KUKA KRL program: MyProgram_299().src

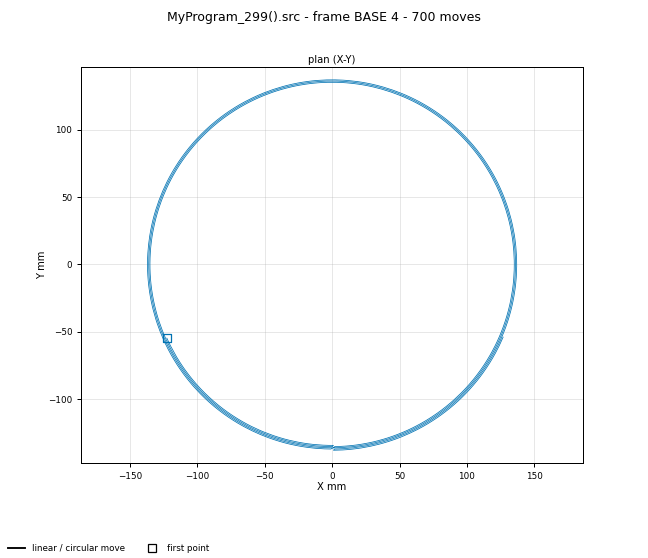
[picture p0: tool path of MyProgram_299().src in frame BASE 4, 700 of 700 moves have a stored position in this frame; points joined in program order, loops and branches not executed]
&ACCESS RVP
&REL 1
&PARAM TEMPLATE = C:\KRC\Roboter\Template\vorgabe
&PARAM EDITMASK = *
DEF MyProgram_299()
; ---- Setting reference (Base) ----
$BASE = BASE_DATA[4]

; --------------------------
; ---- Setting tool (TCP) ----
$TOOL = TOOL_DATA[3]
; --------------------------

$VEL.CP = VEL_APROX_PRINT
Startdeposition()
$VEL.CP = VEL_PRINT
LIN {X -122.5353,Y -54.6728,Z 179,A -152.7629,B 5.8346,C 0.2962,E1 5.6965,E2 244.9953} C_DIS
LIN {X -121.3406,Y -57.2786,Z 179,A -151.1206,B 5.8346,C 0.2952,E1 5.6985,E2 243.3016} C_DIS
LIN {X -119.8803,Y -60.2757,Z 179,A -150.0489,B 5.8343,C 0.3023,E1 5.6998,E2 242.2745} C_DIS
LIN {X -115.3298,Y -68.5828,Z 179,A -145.742,B 5.8339,C 0.3096,E1 5.7057,E2 237.9372} C_DIS
LIN {X -113.093,Y -72.2118,Z 179,A -143.8962,B 5.8337,C 0.3137,E1 5.7084,E2 236.089} C_DIS
LIN {X -110.7158,Y -75.8062,Z 179,A -142.321,B 5.8333,C 0.3206,E1 5.7108,E2 234.5476} C_DIS
LIN {X -108.9586,Y -78.3114,Z 179,A -140.8156,B 5.8333,C 0.3216,E1 5.7133,E2 233.0179} C_DIS
LIN {X -106.2267,Y -81.9786,Z 179,A -138.6816,B 5.8331,C 0.3241,E1 5.7169,E2 230.8619} C_DIS
LIN {X -103.487,Y -85.4109,Z 179,A -136.7855,B 5.8329,C 0.3279,E1 5.7203,E2 228.9638} C_DIS
LIN {X -100.6349,Y -88.7534,Z 179,A -134.8401,B 5.8327,C 0.3311,E1 5.7238,E2 227.0102} C_DIS
LIN {X -97.4615,Y -92.227,Z 179,A -132.8394,B 5.8325,C 0.3352,E1 5.7276,E2 225.0111} C_DIS
LIN {X -94.3505,Y -95.4076,Z 179,A -130.8567,B 5.8323,C 0.3381,E1 5.7316,E2 223.0184} C_DIS
LIN {X -91.2325,Y -98.3933,Z 179,A -129.023,B 5.8321,C 0.3416,E1 5.7353,E2 221.1863} C_DIS
LIN {X -87.9809,Y -101.3114,Z 179,A -127.0949,B 5.832,C 0.3443,E1 5.7393,E2 219.2506} C_DIS
LIN {X -84.7827,Y -104.0022,Z 179,A -125.3045,B 5.8318,C 0.3474,E1 5.7432,E2 217.4598} C_DIS
LIN {X -81.2326,Y -106.7986,Z 179,A -123.3307,B 5.8316,C 0.3501,E1 5.7476,E2 215.4807} C_DIS
LIN {X -77.5555,Y -109.4977,Z 179,A -121.3497,B 5.8314,C 0.3528,E1 5.7521,E2 213.4956} C_DIS
LIN {X -73.9635,Y -111.9552,Z 179,A -119.4643,B 5.8313,C 0.3553,E1 5.7564,E2 211.6069} C_DIS
LIN {X -70.1063,Y -114.41,Z 179,A -117.5715,B 5.8311,C 0.3587,E1 5.7609,E2 209.7217} C_DIS
LIN {X -66.7518,Y -116.3994,Z 179,A -115.8163,B 5.8311,C 0.3599,E1 5.7652,E2 207.9551} C_DIS
LIN {X -63.1485,Y -118.3933,Z 179,A -114.0225,B 5.8309,C 0.3617,E1 5.7696,E2 206.1568} C_DIS
LIN {X -59.718,Y -120.1579,Z 179,A -112.5072,B 5.8307,C 0.3652,E1 5.7733,E2 204.6579} C_DIS
LIN {X -56.4178,Y -121.7417,Z 179,A -110.8814,B 5.8307,C 0.3662,E1 5.7775,E2 203.0241} C_DIS
LIN {X -53.5496,Y -123.0307,Z 179,A -109.5257,B 5.8305,C 0.3674,E1 5.7809,E2 201.6667} C_DIS
LIN {X -50.4662,Y -124.3273,Z 179,A -108.0389,B 5.8305,C 0.3682,E1 5.7848,E2 200.1723} C_DIS
LIN {X -45.7998,Y -126.121,Z 179,A -106.1587,B 5.8302,C 0.3731,E1 5.7896,E2 198.3239} C_DIS
LIN {X -43.4144,Y -126.9628,Z 179,A -104.3015,B 5.8307,C 0.3647,E1 5.7948,E2 196.3679} C_DIS
LIN {X -39.0487,Y -128.3717,Z 179,A -102.5129,B 5.8305,C 0.3681,E1 5.7995,E2 194.6006} C_DIS
LIN {X -35.3556,Y -129.4399,Z 179,A -101.1039,B 5.8303,C 0.372,E1 5.8032,E2 193.2208} C_DIS
LIN {X -31.7308,Y -130.3737,Z 179,A -99.589,B 5.8301,C 0.3739,E1 5.8073,E2 191.7161} C_DIS
LIN {X -28.3423,Y -131.1518,Z 179,A -98.2752,B 5.83,C 0.3768,E1 5.8108,E2 190.4235} C_DIS
LIN {X -25.2631,Y -131.7796,Z 179,A -96.7211,B 5.83,C 0.3747,E1 5.8152,E2 188.8421} C_DIS
LIN {X -20.8136,Y -132.5555,Z 179,A -94.8485,B 5.83,C 0.3761,E1 5.8203,E2 186.9759} C_DIS
LIN {X -17.8111,Y -132.9925,Z 179,A -93.6849,B 5.8299,C 0.3781,E1 5.8235,E2 185.8287} C_DIS
LIN {X -13.6892,Y -133.481,Z 179,A -91.6382,B 5.8301,C 0.375,E1 5.8293,E2 183.7465} C_DIS
LIN {X -9.7537,Y -133.8245,Z 179,A -90.1276,B 5.8299,C 0.3774,E1 5.8334,E2 182.2575} C_DIS
LIN {X -6.6981,Y -134.0122,Z 179,A -88.761,B 5.8299,C 0.3767,E1 5.8372,E2 180.8829} C_DIS
LIN {X -2.5064,Y -134.1564,Z 179,A -86.9364,B 5.8299,C 0.3762,E1 5.8423,E2 179.0532} C_DIS
LIN {X 0.9693,Y -134.1718,Z 179,A -85.948,B 5.8296,C 0.3824,E1 5.845,E2 178.1268} C_DIS
Enddeposition()
LIN {X 0.9693,Y -134.1718,Z 179,A -85.948,B 5.8296,C 0.3824,E1 5.845,E2 178.1268} C_DIS
Startdeposition()
$VEL.CP = VEL_PRINT
LIN {X 0.1925,Y -135.0839,Z 179,A -86.9182,B 5.8288,C 0.3941,E1 5.8419,E2 179.211} C_DIS
LIN {X -3.8541,Y -135.0279,Z 179,A -88.4104,B 5.829,C 0.3913,E1 5.8378,E2 180.6758} C_DIS
LIN {X -8.4195,Y -134.8202,Z 179,A -90.1357,B 5.8292,C 0.3885,E1 5.8331,E2 182.375} C_DIS
LIN {X -11.8698,Y -134.5612,Z 179,A -91.5533,B 5.8292,C 0.3877,E1 5.8291,E2 183.7868} C_DIS
LIN {X -18.7809,Y -133.7711,Z 179,A -94.3462,B 5.8294,C 0.3851,E1 5.8214,E2 186.5609} C_DIS
LIN {X -22.0515,Y -133.2707,Z 179,A -95.9725,B 5.8292,C 0.3874,E1 5.8169,E2 188.2159} C_DIS
LIN {X -25.7307,Y -132.6099,Z 179,A -97.6431,B 5.8292,C 0.3879,E1 5.8122,E2 189.8978} C_DIS
LIN {X -30.1303,Y -131.6794,Z 179,A -99.4733,B 5.8293,C 0.386,E1 5.8073,E2 191.7188} C_DIS
LIN {X -33.2981,Y -130.9142,Z 179,A -100.8597,B 5.8293,C 0.3852,E1 5.8035,E2 193.1061} C_DIS
LIN {X -36.7151,Y -129.9977,Z 179,A -102.3696,B 5.8294,C 0.3844,E1 5.7994,E2 194.6175} C_DIS
LIN {X -39.7924,Y -129.0886,Z 179,A -104.2916,B 5.8291,C 0.3901,E1 5.7941,E2 196.6103} C_DIS
LIN {X -44.2389,Y -127.633,Z 179,A -105.7676,B 5.8296,C 0.3825,E1 5.7904,E2 198.0229} C_DIS
LIN {X -47.8774,Y -126.3143,Z 179,A -107.4013,B 5.8296,C 0.381,E1 5.7861,E2 199.656} C_DIS
LIN {X -50.6962,Y -125.2085,Z 179,A -108.6766,B 5.8297,C 0.3796,E1 5.7828,E2 200.9302} C_DIS
LIN {X -53.8918,Y -123.8669,Z 179,A -110.1441,B 5.8298,C 0.3781,E1 5.779,E2 202.3976} C_DIS
LIN {X -56.8726,Y -122.5266,Z 179,A -111.571,B 5.8299,C 0.3771,E1 5.7754,E2 203.8298} C_DIS
LIN {X -60.0173,Y -121.0175,Z 179,A -113.0316,B 5.83,C 0.3752,E1 5.7717,E2 205.288} C_DIS
LIN {X -63.4706,Y -119.2446,Z 179,A -114.7609,B 5.8301,C 0.3741,E1 5.7674,E2 207.028} C_DIS
LIN {X -67.2872,Y -117.134,Z 179,A -116.7066,B 5.8301,C 0.3728,E1 5.7627,E2 208.9857} C_DIS
LIN {X -71.0224,Y -114.9075,Z 179,A -118.586,B 5.8303,C 0.3706,E1 5.7582,E2 210.8695} C_DIS
LIN {X -74.8806,Y -112.4308,Z 179,A -120.5246,B 5.8305,C 0.3677,E1 5.7536,E2 212.8073} C_DIS
LIN {X -78.7391,Y -109.7632,Z 179,A -122.5421,B 5.8307,C 0.3649,E1 5.749,E2 214.8281} C_DIS
LIN {X -82.3408,Y -107.0882,Z 179,A -124.4845,B 5.8308,C 0.3623,E1 5.7447,E2 216.7753} C_DIS
LIN {X -85.6454,Y -104.4638,Z 179,A -126.2751,B 5.831,C 0.3592,E1 5.7408,E2 218.5657} C_DIS
LIN {X -89.0754,Y -101.5552,Z 179,A -128.2265,B 5.8312,C 0.3563,E1 5.7366,E2 220.5224} C_DIS
LIN {X -92.4123,Y -98.5286,Z 179,A -130.1861,B 5.8314,C 0.3533,E1 5.7326,E2 222.4877} C_DIS
LIN {X -95.6095,Y -95.4289,Z 179,A -132.1017,B 5.8316,C 0.3499,E1 5.7288,E2 224.4062} C_DIS
LIN {X -98.7676,Y -92.1561,Z 179,A -134.2548,B 5.8316,C 0.3484,E1 5.7246,E2 226.5867} C_DIS
LIN {X -100.9945,Y -89.7105,Z 179,A -135.3308,B 5.8321,C 0.3421,E1 5.7227,E2 227.6216} C_DIS
LIN {X -103.3298,Y -87.0103,Z 179,A -137.0372,B 5.8321,C 0.3409,E1 5.7195,E2 229.3515} C_DIS
LIN {X -106.1821,Y -83.5054,Z 179,A -138.9727,B 5.8324,C 0.3369,E1 5.7162,E2 231.2888} C_DIS
LIN {X -109.0769,Y -79.6876,Z 179,A -141.0485,B 5.8326,C 0.3328,E1 5.7127,E2 233.3693} C_DIS
LIN {X -111.6524,Y -76.0372,Z 179,A -142.8629,B 5.8329,C 0.3277,E1 5.7098,E2 235.1729} C_DIS
LIN {X -113.7398,Y -72.8768,Z 179,A -144.6262,B 5.833,C 0.3255,E1 5.7071,E2 236.955} C_DIS
LIN {X -116.2063,Y -68.8765,Z 179,A -146.9133,B 5.8331,C 0.3236,E1 5.7037,E2 239.2777} C_DIS
LIN {X -117.9348,Y -65.8712,Z 179,A -148.5238,B 5.8332,C 0.3214,E1 5.7015,E2 240.9047} C_DIS
LIN {X -119.8665,Y -62.2862,Z 179,A -149.8352,B 5.8337,C 0.313,E1 5.6999,E2 242.1639} C_DIS
LIN {X -121.8462,Y -58.3159,Z 179,A -151.6473,B 5.834,C 0.3076,E1 5.6977,E2 243.9664} C_DIS
LIN {X -122.8584,Y -56.1552,Z 179,A -152.7758,B 5.834,C 0.3062,E1 5.6963,E2 245.1089} C_DIS
LIN {X -124.4198,Y -52.6052,Z 179,A -154.548,B 5.8342,C 0.3031,E1 5.6944,E2 246.896} C_DIS
LIN {X -125.9347,Y -48.864,Z 179,A -156.6034,B 5.8342,C 0.3019,E1 5.6922,E2 248.9927} C_DIS
LIN {X -127.2364,Y -45.3695,Z 179,A -157.7965,B 5.8347,C 0.294,E1 5.6911,E2 250.1371} C_DIS
LIN {X -128.1949,Y -42.5834,Z 179,A -159.1541,B 5.8347,C 0.2917,E1 5.6899,E2 251.5072} C_DIS
LIN {X -129.4006,Y -38.7733,Z 179,A -160.951,B 5.835,C 0.2881,E1 5.6884,E2 253.3157} C_DIS
LIN {X -130.3952,Y -35.2793,Z 179,A -163.1042,B 5.8349,C 0.2897,E1 5.6868,E2 255.5428} C_DIS
LIN {X -131.6356,Y -30.3223,Z 179,A -164.4239,B 5.8356,C 0.2757,E1 5.686,E2 256.7572} C_DIS
LIN {X -132.4516,Y -26.534,Z 179,A -166.3905,B 5.8356,C 0.2742,E1 5.6848,E2 258.7625} C_DIS
LIN {X -133.2044,Y -22.4492,Z 179,A -168.2053,B 5.8358,C 0.2697,E1 5.684,E2 260.5826} C_DIS
LIN {X -133.8225,Y -18.4214,Z 179,A -170.0707,B 5.836,C 0.2662,E1 5.6832,E2 262.4637} C_DIS
LIN {X -134.3063,Y -14.4627,Z 179,A -171.6632,B 5.8363,C 0.2605,E1 5.6827,E2 264.0427} C_DIS
LIN {X -134.6447,Y -10.8814,Z 179,A -173.3305,B 5.8363,C 0.2575,E1 5.6823,E2 265.7262} C_DIS
LIN {X -134.9116,Y -6.7998,Z 179,A -174.9866,B 5.8366,C 0.2518,E1 5.682,E2 267.3714} C_DIS
LIN {X -135.0465,Y -3.1856,Z 179,A -176.6927,B 5.8368,C 0.249,E1 5.6819,E2 269.0974} C_DIS
LIN {X -135.0815,Y 0.77,Z 179,A -178.319,B 5.837,C 0.2437,E1 5.6819,E2 270.7161} C_DIS
LIN {X -134.9975,Y 4.8204,Z 179,A 179.8767,B 5.8372,C 0.2396,E1 5.682,E2 272.5295} C_DIS
LIN {X -134.7986,Y 8.7696,Z 179,A 178.1435,B 5.8373,C 0.2354,E1 5.6823,E2 274.2682} C_DIS
LIN {X -134.4785,Y 12.7631,Z 179,A 176.4737,B 5.8375,C 0.2303,E1 5.6827,E2 275.933} C_DIS
LIN {X -134.1088,Y 16.1925,Z 179,A 174.9726,B 5.8377,C 0.2265,E1 5.6832,E2 277.4376} C_DIS
LIN {X -133.5512,Y 20.287,Z 179,A 173.1379,B 5.8378,C 0.2223,E1 5.6839,E2 279.2807} C_DIS
LIN {X -132.9852,Y 23.7123,Z 179,A 171.6967,B 5.838,C 0.2178,E1 5.6846,E2 280.7169} C_DIS
LIN {X -132.31,Y 27.2297,Z 179,A 170.1203,B 5.8381,C 0.2141,E1 5.6854,E2 282.2989} C_DIS
LIN {X -131.6394,Y 30.3053,Z 179,A 168.7103,B 5.8383,C 0.2111,E1 5.6863,E2 283.7169} C_DIS
LIN {X -130.6958,Y 34.1519,Z 179,A 167.0743,B 5.8384,C 0.206,E1 5.6874,E2 285.3462} C_DIS
LIN {X -129.5807,Y 38.1597,Z 179,A 165.217,B 5.8386,C 0.202,E1 5.6888,E2 287.2131} C_DIS
LIN {X -128.4802,Y 41.7197,Z 179,A 163.6139,B 5.8387,C 0.1979,E1 5.6902,E2 288.8177} C_DIS
LIN {X -126.6284,Y 47.0385,Z 179,A 161.3378,B 5.839,C 0.1904,E1 5.6923,E2 291.078} C_DIS
LIN {X -125.1791,Y 50.7693,Z 179,A 159.3995,B 5.839,C 0.1882,E1 5.6943,E2 293.044} C_DIS
LIN {X -123.7336,Y 54.2001,Z 179,A 157.8119,B 5.8392,C 0.1841,E1 5.696,E2 294.6313} C_DIS
LIN {X -122.5017,Y 56.9265,Z 179,A 156.5211,B 5.8392,C 0.181,E1 5.6975,E2 295.9234} C_DIS
LIN {X -121.2322,Y 59.5819,Z 179,A 154.7765,B 5.8392,C 0.1825,E1 5.6998,E2 297.7267} C_DIS
LIN {X -119.4113,Y 63.1531,Z 179,A 153.6102,B 5.8395,C 0.1731,E1 5.7012,E2 298.8273} C_DIS
LIN {X -117.6163,Y 66.4399,Z 179,A 151.7431,B 5.8395,C 0.1718,E1 5.7037,E2 300.7266} C_DIS
LIN {X -115.207,Y 70.5346,Z 179,A 149.4802,B 5.8396,C 0.1693,E1 5.707,E2 303.0175} C_DIS
LIN {X -113.4269,Y 73.3632,Z 179,A 148.1994,B 5.8397,C 0.1646,E1 5.709,E2 304.2806} C_DIS
LIN {X -111.0661,Y 76.8908,Z 179,A 146.3786,B 5.8399,C 0.1605,E1 5.7118,E2 306.1022} C_DIS
LIN {X -108.3594,Y 80.6598,Z 179,A 144.4191,B 5.8399,C 0.1559,E1 5.715,E2 308.059} C_DIS
LIN {X -105.5992,Y 84.2413,Z 179,A 142.4693,B 5.8401,C 0.1519,E1 5.7184,E2 310.0109} C_DIS
LIN {X -102.7629,Y 87.6791,Z 179,A 140.5494,B 5.8401,C 0.1481,E1 5.7219,E2 311.9327} C_DIS
LIN {X -100.0781,Y 90.7311,Z 179,A 138.772,B 5.8403,C 0.1449,E1 5.7252,E2 313.715} C_DIS
LIN {X -97.1859,Y 93.8227,Z 179,A 136.9148,B 5.8403,C 0.1418,E1 5.7288,E2 315.578} C_DIS
LIN {X -93.9282,Y 97.0838,Z 179,A 134.9532,B 5.8404,C 0.138,E1 5.7327,E2 317.5387} C_DIS
LIN {X -90.573,Y 100.2216,Z 179,A 132.9754,B 5.8405,C 0.1345,E1 5.7367,E2 319.5183} C_DIS
LIN {X -87.3475,Y 103.0448,Z 179,A 131.1131,B 5.8405,C 0.1316,E1 5.7407,E2 321.3844} C_DIS
LIN {X -83.8167,Y 105.9372,Z 179,A 129.1345,B 5.8406,C 0.1286,E1 5.745,E2 323.3665} C_DIS
LIN {X -80.3697,Y 108.5754,Z 179,A 127.2618,B 5.8407,C 0.1258,E1 5.7492,E2 325.2415} C_DIS
LIN {X -76.7484,Y 111.1647,Z 179,A 125.3623,B 5.8407,C 0.1229,E1 5.7535,E2 327.1408} C_DIS
LIN {X -71.9992,Y 114.2972,Z 179,A 122.4982,B 5.8407,C 0.1239,E1 5.7604,E2 330.0566} C_DIS
LIN {X -68.2451,Y 116.578,Z 179,A 121.196,B 5.8409,C 0.1153,E1 5.7633,E2 331.2906} C_DIS
LIN {X -64.4385,Y 118.7246,Z 179,A 118.9099,B 5.8409,C 0.1174,E1 5.769,E2 333.6269} C_DIS
LIN {X -61.5238,Y 120.2585,Z 179,A 118.0579,B 5.841,C 0.1097,E1 5.771,E2 334.4127} C_DIS
LIN {X -57.8524,Y 122.0676,Z 179,A 116.0801,B 5.841,C 0.1102,E1 5.776,E2 336.4183} C_DIS
LIN {X -54.1238,Y 123.7666,Z 179,A 114.1375,B 5.841,C 0.1105,E1 5.781,E2 338.384} C_DIS
LIN {X -50.3061,Y 125.3658,Z 179,A 111.6949,B 5.841,C 0.1162,E1 5.7876,E2 340.9065} C_DIS
LIN {X -44.5114,Y 127.5385,Z 179,A 109.848,B 5.8411,C 0.1051,E1 5.7922,E2 342.6598} C_DIS
LIN {X -41.8008,Y 128.4543,Z 179,A 108.4722,B 5.8411,C 0.1059,E1 5.7959,E2 344.0541} C_DIS
LIN {X -37.5588,Y 129.7566,Z 179,A 106.8419,B 5.8411,C 0.1016,E1 5.8002,E2 345.6533} C_DIS
LIN {X -34.5569,Y 130.5878,Z 179,A 105.4059,B 5.8411,C 0.1019,E1 5.8041,E2 347.102} C_DIS
LIN {X -30.3229,Y 131.6354,Z 179,A 103.5321,B 5.8411,C 0.101,E1 5.8092,E2 348.9775} C_DIS
LIN {X -26.856,Y 132.3861,Z 179,A 102.1376,B 5.8412,C 0.0989,E1 5.8129,E2 350.3581} C_DIS
LIN {X -23.5734,Y 133.01,Z 179,A 100.6014,B 5.8412,C 0.0996,E1 5.8172,E2 351.9076} C_DIS
LIN {X -19.237,Y 133.706,Z 179,A 98.7616,B 5.8412,C 0.0986,E1 5.8223,E2 353.7437} C_DIS
LIN {X -15.2247,Y 134.2242,Z 179,A 96.4643,B 5.8412,C 0.1049,E1 5.8288,E2 356.1091} C_DIS
LIN {X -10.4045,Y 134.6827,Z 179,A 95.1103,B 5.8412,C 0.0962,E1 5.8324,E2 357.3789} C_DIS
LIN {X -6.7031,Y 134.9164,Z 179,A 93.4283,B 5.8412,C 0.0973,E1 5.8371,E2 359.0732} C_DIS
LIN {X -3.24,Y 135.045,Z 179,A 91.6532,B 5.8412,C 0.1009,E1 5.8421,E2 360.884} C_DIS
LIN {X 0.0997,Y 135.0836,Z 179,A 90.2647,B 5.8412,C 0.1006,E1 5.846,E2 362.2685} C_DIS
LIN {X 3.3111,Y 135.043,Z 179,A 89.1887,B 5.8412,C 0.0972,E1 5.8489,E2 363.3098} C_DIS
LIN {X 6.7159,Y 134.9158,Z 179,A 87.7255,B 5.8412,C 0.0977,E1 5.853,E2 364.7746} C_DIS
LIN {X 10.6226,Y 134.6665,Z 179,A 85.5538,B 5.8412,C 0.1044,E1 5.8592,E2 367.0065} C_DIS
LIN {X 15.1065,Y 134.237,Z 179,A 84.2646,B 5.8412,C 0.0973,E1 5.8626,E2 368.2212} C_DIS
LIN {X 19.2325,Y 133.7066,Z 179,A 82.4527,B 5.8412,C 0.0986,E1 5.8676,E2 370.0381} C_DIS
LIN {X 22.386,Y 133.2149,Z 179,A 81.071,B 5.8412,C 0.0996,E1 5.8714,E2 371.4227} C_DIS
LIN {X 26.323,Y 132.4945,Z 179,A 79.254,B 5.8412,C 0.1021,E1 5.8765,E2 373.2535} C_DIS
LIN {X 30.4729,Y 131.6012,Z 179,A 77.6339,B 5.8412,C 0.1009,E1 5.8808,E2 374.8516} C_DIS
LIN {X 33.5262,Y 130.8563,Z 179,A 76.2571,B 5.8412,C 0.1025,E1 5.8846,E2 376.2332} C_DIS
LIN {X 36.6147,Y 130.0256,Z 179,A 74.3524,B 5.841,C 0.1107,E1 5.8899,E2 378.203} C_DIS
LIN {X 41.1601,Y 128.6589,Z 179,A 73.2687,B 5.8412,C 0.1002,E1 5.8925,E2 379.1752} C_DIS
LIN {X 43.8876,Y 127.7548,Z 179,A 71.6861,B 5.8411,C 0.1062,E1 5.8968,E2 380.8013} C_DIS
LIN {X 47.7005,Y 126.3805,Z 179,A 70.0437,B 5.8411,C 0.1069,E1 5.901,E2 382.4343} C_DIS
LIN {X 50.5566,Y 125.2648,Z 179,A 68.7199,B 5.8411,C 0.1086,E1 5.9045,E2 383.7607} C_DIS
LIN {X 53.6379,Y 123.9766,Z 179,A 67.2929,B 5.8411,C 0.1104,E1 5.9082,E2 385.1888} C_DIS
LIN {X 56.8746,Y 122.5257,Z 179,A 65.8366,B 5.841,C 0.1115,E1 5.9118,E2 386.6392} C_DIS
LIN {X 60.0247,Y 121.0138,Z 179,A 64.3619,B 5.841,C 0.1133,E1 5.9155,E2 388.113} C_DIS
LIN {X 63.1268,Y 119.4251,Z 179,A 62.8766,B 5.841,C 0.1154,E1 5.9192,E2 389.599} C_DIS
LIN {X 66.8787,Y 117.367,Z 179,A 61.071,B 5.8409,C 0.1178,E1 5.9236,E2 391.4035} C_DIS
LIN {X 70.4681,Y 115.2478,Z 179,A 59.3279,B 5.8409,C 0.1201,E1 5.9278,E2 393.1436} C_DIS
LIN {X 73.7387,Y 113.1831,Z 179,A 57.6929,B 5.8408,C 0.1226,E1 5.9316,E2 394.778} C_DIS
LIN {X 77.3792,Y 110.7263,Z 179,A 55.8391,B 5.8408,C 0.1255,E1 5.9359,E2 396.6309} C_DIS
LIN {X 80.9825,Y 108.1191,Z 179,A 53.9266,B 5.8406,C 0.1291,E1 5.9402,E2 398.5467} C_DIS
LIN {X 84.5024,Y 105.391,Z 179,A 52.0582,B 5.8406,C 0.1321,E1 5.9443,E2 400.4129} C_DIS
LIN {X 88.0294,Y 102.4627,Z 179,A 50.1749,B 5.8406,C 0.1349,E1 5.9483,E2 402.2891} C_DIS
LIN {X 93.1247,Y 97.8552,Z 179,A 47.4734,B 5.8404,C 0.1375,E1 5.9538,E2 404.9655} C_DIS
LIN {X 95.6611,Y 95.377,Z 179,A 45.524,B 5.8402,C 0.147,E1 5.9578,E2 406.969} C_DIS
LIN {X 98.396,Y 92.5529,Z 179,A 44.3056,B 5.8402,C 0.1439,E1 5.96,E2 408.1337} C_DIS
LIN {X 101.0076,Y 89.6957,Z 179,A 42.5662,B 5.8402,C 0.1488,E1 5.9633,E2 409.8853} C_DIS
LIN {X 104.2929,Y 85.854,Z 179,A 40.4618,B 5.8401,C 0.1529,E1 5.9671,E2 411.9856} C_DIS
LIN {X 107.3685,Y 81.9743,Z 179,A 38.6251,B 5.8401,C 0.1537,E1 5.9702,E2 413.791} C_DIS
LIN {X 109.5483,Y 79.0382,Z 179,A 36.9492,B 5.8399,C 0.1591,E1 5.973,E2 415.4827} C_DIS
LIN {X 111.8758,Y 75.7072,Z 179,A 35.2687,B 5.8398,C 0.1625,E1 5.9756,E2 417.1586} C_DIS
LIN {X 114.2113,Y 72.1357,Z 179,A 33.4497,B 5.8397,C 0.167,E1 5.9784,E2 418.9795} C_DIS
LIN {X 116.6028,Y 68.2029,Z 179,A 31.5617,B 5.8396,C 0.1708,E1 5.9811,E2 420.8604} C_DIS
LIN {X 118.7744,Y 64.3472,Z 179,A 29.6813,B 5.8394,C 0.1756,E1 5.9836,E2 422.7421} C_DIS
LIN {X 120.6863,Y 60.6836,Z 179,A 28.102,B 5.8394,C 0.1774,E1 5.9856,E2 424.3011} C_DIS
LIN {X 121.9825,Y 58.0305,Z 179,A 26.8288,B 5.8393,C 0.1809,E1 5.9872,E2 425.5774} C_DIS
LIN {X 123.6846,Y 54.3135,Z 179,A 24.8879,B 5.839,C 0.1886,E1 5.9894,E2 427.5445} C_DIS
LIN {X 125.9,Y 48.9533,Z 179,A 22.679,B 5.839,C 0.1912,E1 5.9917,E2 429.724} C_DIS
LIN {X 127.3149,Y 45.1517,Z 179,A 20.9581,B 5.8388,C 0.1958,E1 5.9933,E2 431.446} C_DIS
LIN {X 128.7974,Y 40.7267,Z 179,A 19.1672,B 5.8387,C 0.1983,E1 5.9949,E2 433.2149} C_DIS
LIN {X 129.662,Y 37.882,Z 179,A 17.9236,B 5.8386,C 0.2015,E1 5.9958,E2 434.4571} C_DIS
LIN {X 130.5523,Y 34.6902,Z 179,A 16.5358,B 5.8385,C 0.205,E1 5.9969,E2 435.8436} C_DIS
LIN {X 131.3904,Y 31.3677,Z 179,A 15.1091,B 5.8383,C 0.2087,E1 5.9978,E2 437.268} C_DIS
LIN {X 132.1551,Y 27.9754,Z 179,A 13.5712,B 5.8382,C 0.2137,E1 5.9987,E2 438.8147} C_DIS
LIN {X 132.9492,Y 23.913,Z 179,A 11.9273,B 5.838,C 0.2169,E1 5.9996,E2 440.446} C_DIS
LIN {X 133.5724,Y 20.15,Z 179,A 10.3952,B 5.838,C 0.2201,E1 6.0002,E2 441.9687} C_DIS
LIN {X 134.1297,Y 16.0175,Z 179,A 8.6489,B 5.8377,C 0.2248,E1 6.0009,E2 443.7134} C_DIS
LIN {X 134.508,Y 12.4559,Z 179,A 7.2309,B 5.8377,C 0.2275,E1 6.0013,E2 445.12} C_DIS
LIN {X 134.7387,Y 9.6376,Z 179,A 5.7152,B 5.8373,C 0.2359,E1 6.0016,E2 446.6756} C_DIS
LIN {X 134.936,Y 6.3133,Z 179,A 4.3526,B 5.8372,C 0.2391,E1 6.0018,E2 448.0332} C_DIS
LIN {X 135.0508,Y 3.0322,Z 179,A 3.3079,B 5.8372,C 0.2377,E1 6.0018,E2 449.0361} C_DIS
LIN {X 135.0857,Y -0.0693,Z 179,A 1.8506,B 5.837,C 0.2436,E1 6.0018,E2 450.512} C_DIS
LIN {X 135.0142,Y -4.3482,Z 179,A -0.6217,B 5.8363,C 0.2591,E1 6.0016,E2 453.0664} C_DIS
LIN {X 134.6676,Y -10.6108,Z 179,A -2.5425,B 5.8365,C 0.2551,E1 6.0013,E2 454.8985} C_DIS
LIN {X 134.239,Y -15.0879,Z 179,A -4.3805,B 5.8363,C 0.2595,E1 6.0007,E2 456.7294} C_DIS
LIN {X 133.7286,Y -19.0788,Z 179,A -5.8928,B 5.8363,C 0.2613,E1 6.0002,E2 458.219} C_DIS
LIN {X 132.8937,Y -24.2236,Z 179,A -7.9642,B 5.836,C 0.2653,E1 5.9992,E2 460.275} C_DIS
LIN {X 132.3745,Y -26.9126,Z 179,A -9.2413,B 5.8358,C 0.2704,E1 5.9985,E2 461.5674} C_DIS
LIN {X 131.6534,Y -30.2444,Z 179,A -10.625,B 5.8357,C 0.2735,E1 5.9977,E2 462.9446} C_DIS
LIN {X 130.699,Y -34.1399,Z 179,A -12.5296,B 5.8353,C 0.2814,E1 5.9964,E2 464.876} C_DIS
LIN {X 129.5423,Y -38.2909,Z 179,A -14.0717,B 5.8353,C 0.282,E1 5.9952,E2 466.3842} C_DIS
LIN {X 128.3605,Y -42.086,Z 179,A -16.1727,B 5.8347,C 0.2931,E1 5.9933,E2 468.5383} C_DIS
LIN {X 127.002,Y -46.0194,Z 179,A -17.3187,B 5.835,C 0.2882,E1 5.9923,E2 469.6086} C_DIS
LIN {X 125.1985,Y -50.7211,Z 179,A -19.5038,B 5.8346,C 0.2947,E1 5.9901,E2 471.802} C_DIS
LIN {X 123.9655,Y -53.6636,Z 179,A -20.874,B 5.8344,C 0.2986,E1 5.9886,E2 473.1755} C_DIS
LIN {X 122.5163,Y -56.895,Z 179,A -22.3223,B 5.8343,C 0.3017,E1 5.9869,E2 474.6184} C_DIS
LIN {X 121.0717,Y -59.9074,Z 179,A -24.3764,B 5.8336,C 0.3152,E1 5.9843,E2 476.7532} C_DIS
LIN {X 118.5283,Y -64.7984,Z 179,A -25.8527,B 5.834,C 0.3079,E1 5.9825,E2 478.1242} C_DIS
LIN {X 116.8303,Y -67.8121,Z 179,A -27.4882,B 5.8336,C 0.3142,E1 5.9802,E2 479.7821} C_DIS
LIN {X 114.7252,Y -71.3156,Z 179,A -29.1791,B 5.8334,C 0.3179,E1 5.9777,E2 481.4692} C_DIS
LIN {X 112.4294,Y -74.8827,Z 179,A -30.9715,B 5.8332,C 0.3221,E1 5.975,E2 483.2624} C_DIS
LIN {X 109.9582,Y -78.4664,Z 179,A -32.7821,B 5.833,C 0.326,E1 5.9721,E2 485.0702} C_DIS
LIN {X 107.1859,Y -82.213,Z 179,A -34.6557,B 5.8328,C 0.329,E1 5.969,E2 486.9326} C_DIS
LIN {X 104.5489,Y -85.5413,Z 179,A -36.4649,B 5.8326,C 0.3333,E1 5.9658,E2 488.7444} C_DIS
LIN {X 101.6303,Y -88.9894,Z 179,A -38.4742,B 5.8322,C 0.339,E1 5.9621,E2 490.7672} C_DIS
LIN {X 99.0454,Y -91.8578,Z 179,A -39.9808,B 5.8322,C 0.3405,E1 5.9593,E2 492.2588} C_DIS
LIN {X 95.926,Y -95.1104,Z 179,A -41.8387,B 5.832,C 0.3438,E1 5.9557,E2 494.1116} C_DIS
LIN {X 90.2898,Y -100.4767,Z 179,A -44.8089,B 5.8319,C 0.3455,E1 5.9497,E2 497.043} C_DIS
LIN {X 88.0647,Y -102.4323,Z 179,A -46.318,B 5.8315,C 0.3517,E1 5.9465,E2 498.5852} C_DIS
LIN {X 84.5411,Y -105.3598,Z 179,A -48.2318,B 5.8313,C 0.355,E1 5.9423,E2 500.497} C_DIS
LIN {X 81.226,Y -107.9359,Z 179,A -49.9726,B 5.8311,C 0.3576,E1 5.9385,E2 502.2342} C_DIS
LIN {X 77.6356,Y -110.5467,Z 179,A -51.8665,B 5.8309,C 0.3611,E1 5.9342,E2 504.1311} C_DIS
LIN {X 73.8615,Y -113.1034,Z 179,A -53.7641,B 5.8308,C 0.3638,E1 5.9298,E2 506.0257} C_DIS
LIN {X 70.1305,Y -115.4537,Z 179,A -55.6217,B 5.8306,C 0.3666,E1 5.9254,E2 507.8833} C_DIS
LIN {X 66.04,Y -117.8411,Z 179,A -57.5676,B 5.8304,C 0.3687,E1 5.9207,E2 509.8228} C_DIS
LIN {X 62.3383,Y -119.8392,Z 179,A -59.3276,B 5.8304,C 0.3709,E1 5.9163,E2 511.5811} C_DIS
LIN {X 59.2347,Y -121.4036,Z 179,A -60.6906,B 5.8303,C 0.3714,E1 5.9129,E2 512.9311} C_DIS
LIN {X 55.9487,Y -122.9539,Z 179,A -62.2216,B 5.8302,C 0.3732,E1 5.9091,E2 514.462} C_DIS
LIN {X 52.9181,Y -124.2879,Z 179,A -64.2025,B 5.8295,C 0.3831,E1 5.9038,E2 516.5167} C_DIS
LIN {X 48.4641,Y -126.0902,Z 179,A -65.637,B 5.8299,C 0.377,E1 5.9003,E2 517.8766} C_DIS
LIN {X 44.5125,Y -127.5381,Z 179,A -67.5055,B 5.8297,C 0.3801,E1 5.8953,E2 519.7569} C_DIS
LIN {X 40.9857,Y -128.7146,Z 179,A -68.9676,B 5.8297,C 0.3801,E1 5.8915,E2 521.2055} C_DIS
LIN {X 37.7273,Y -129.7073,Z 179,A -70.4329,B 5.8297,C 0.3817,E1 5.8875,E2 522.6745} C_DIS
LIN {X 33.4918,Y -130.8651,Z 179,A -72.2704,B 5.8295,C 0.3829,E1 5.8826,E2 524.5101} C_DIS
LIN {X 29.9456,Y -131.7216,Z 179,A -73.7639,B 5.8295,C 0.3834,E1 5.8785,E2 525.9977} C_DIS
LIN {X 26.7335,Y -132.411,Z 179,A -75.2045,B 5.8294,C 0.385,E1 5.8746,E2 527.4451} C_DIS
LIN {X 21.7028,Y -133.3289,Z 179,A -77.2348,B 5.8294,C 0.3845,E1 5.869,E2 529.4592} C_DIS
LIN {X 17.6161,Y -133.9291,Z 179,A -79.0549,B 5.8294,C 0.3863,E1 5.864,E2 531.2889} C_DIS
LIN {X 14.3575,Y -134.3176,Z 179,A -80.871,B 5.8289,C 0.3925,E1 5.8588,E2 533.1593} C_DIS
LIN {X 10.4047,Y -134.6822,Z 179,A -82.3701,B 5.829,C 0.3907,E1 5.8547,E2 534.6361} C_DIS
LIN {X 5.7059,Y -134.963,Z 179,A -84.1772,B 5.8291,C 0.3887,E1 5.8497,E2 536.4203} C_DIS
LIN {X 2.0456,Y -135.0676,Z 179,A -85.6764,B 5.8291,C 0.3883,E1 5.8455,E2 537.9134} C_DIS
LIN {X 2.0456,Y -135.0676,Z 179,A -85.6764,B 5.8291,C 0.3883,E1 5.8455,E2 537.9134} C_DIS
Enddeposition()
LIN {X 0.9634,Y -135.9823,Z 179,A -86.8695,B 5.7039,C 0.3997,E1 5.7175,E2 539.2684} C_DIS
Startdeposition()
$VEL.CP = VEL_PRINT
LIN {X 8.0501,Y -135.748,Z 179,A -82.6268,B 5.7051,C 0.3831,E1 5.7298,E2 534.8647} C_DIS
LIN {X 15.2055,Y -135.1349,Z 179,A -79.2776,B 5.7054,C 0.3776,E1 5.7392,E2 531.4723} C_DIS
LIN {X 18.2105,Y -134.7623,Z 179,A -77.9507,B 5.7055,C 0.3763,E1 5.7429,E2 530.1381} C_DIS
LIN {X 23.6983,Y -133.9053,Z 179,A -75.7848,B 5.7055,C 0.3773,E1 5.7488,E2 527.9934} C_DIS
LIN {X 27.5667,Y -133.1633,Z 179,A -74.0325,B 5.7056,C 0.3749,E1 5.7537,E2 526.2281} C_DIS
LIN {X 31.3928,Y -132.3136,Z 179,A -72.4598,B 5.7056,C 0.3747,E1 5.7579,E2 524.6645} C_DIS
LIN {X 34.7009,Y -131.4843,Z 179,A -71.0492,B 5.7056,C 0.3739,E1 5.7617,E2 523.2563} C_DIS
LIN {X 38.2301,Y -130.5013,Z 179,A -69.6136,B 5.7056,C 0.3739,E1 5.7656,E2 521.8337} C_DIS
LIN {X 41.1477,Y -129.6112,Z 179,A -68.3298,B 5.7057,C 0.3728,E1 5.769,E2 520.5492} C_DIS
LIN {X 45.2284,Y -128.2458,Z 179,A -66.5182,B 5.7059,C 0.3709,E1 5.7738,E2 518.7365} C_DIS
LIN {X 51.3938,Y -125.9013,Z 179,A -63.5035,B 5.7063,C 0.3644,E1 5.7817,E2 515.6895} C_DIS
LIN {X 55.4813,Y -124.1528,Z 179,A -61.929,B 5.7062,C 0.3663,E1 5.7856,E2 514.1522} C_DIS
LIN {X 58.1908,Y -122.9071,Z 179,A -60.5311,B 5.7064,C 0.3626,E1 5.7892,E2 512.7351} C_DIS
LIN {X 61.4791,Y -121.2949,Z 179,A -59.1484,B 5.7064,C 0.3628,E1 5.7926,E2 511.3719} C_DIS
LIN {X 64.8414,Y -119.5338,Z 179,A -57.4315,B 5.7066,C 0.3588,E1 5.7969,E2 509.6387} C_DIS
LIN {X 68.6771,Y -117.3718,Z 179,A -55.6004,B 5.7068,C 0.3563,E1 5.8013,E2 507.8092} C_DIS
LIN {X 72.6429,Y -114.9594,Z 179,A -53.7148,B 5.7069,C 0.3542,E1 5.8058,E2 505.931} C_DIS
LIN {X 76.3001,Y -112.5653,Z 179,A -51.8697,B 5.7071,C 0.3511,E1 5.8101,E2 504.084} C_DIS
LIN {X 80.1127,Y -109.8852,Z 179,A -49.92,B 5.7073,C 0.3479,E1 5.8145,E2 502.1344} C_DIS
LIN {X 83.6835,Y -107.1908,Z 179,A -48.0468,B 5.7075,C 0.3446,E1 5.8187,E2 500.2611} C_DIS
LIN {X 87.2581,Y -104.301,Z 179,A -46.1683,B 5.7077,C 0.3418,E1 5.8227,E2 498.3885} C_DIS
LIN {X 90.6818,Y -101.3383,Z 179,A -44.3843,B 5.7077,C 0.3399,E1 5.8264,E2 496.6188} C_DIS
LIN {X 95.5368,Y -96.7757,Z 179,A -41.5178,B 5.7082,C 0.3333,E1 5.8322,E2 493.7422} C_DIS
LIN {X 98.6757,Y -93.5728,Z 179,A -39.6323,B 5.7084,C 0.3293,E1 5.8359,E2 491.8556} C_DIS
LIN {X 102.0209,Y -89.9134,Z 179,A -37.6423,B 5.7086,C 0.3263,E1 5.8396,E2 489.8765} C_DIS
LIN {X 104.8924,Y -86.5464,Z 179,A -35.8166,B 5.7088,C 0.3227,E1 5.8428,E2 488.0542} C_DIS
LIN {X 107.6848,Y -83.0466,Z 179,A -33.956,B 5.709,C 0.3187,E1 5.846,E2 486.1952} C_DIS
LIN {X 110.3748,Y -79.4369,Z 179,A -32.0899,B 5.7092,C 0.3147,E1 5.8491,E2 484.3313} C_DIS
LIN {X 112.8003,Y -75.9528,Z 179,A -30.4376,B 5.7094,C 0.3125,E1 5.8517,E2 482.6949} C_DIS
LIN {X 115.0499,Y -72.4995,Z 179,A -28.7257,B 5.7096,C 0.3086,E1 5.8543,E2 480.9846} C_DIS
LIN {X 117.1172,Y -69.1107,Z 179,A -27.0026,B 5.7098,C 0.3037,E1 5.8567,E2 479.2534} C_DIS
LIN {X 119.3975,Y -65.0913,Z 179,A -24.948,B 5.7102,C 0.2971,E1 5.8595,E2 477.1832} C_DIS
LIN {X 122.2041,Y -59.6537,Z 179,A -22.6166,B 5.7103,C 0.2942,E1 5.8624,E2 474.8812} C_DIS
LIN {X 123.862,Y -56.1315,Z 179,A -21.0387,B 5.7105,C 0.2909,E1 5.8643,E2 473.3098} C_DIS
LIN {X 125.6199,Y -52.0757,Z 179,A -18.9581,B 5.7109,C 0.2825,E1 5.8666,E2 471.1995} C_DIS
LIN {X 126.8969,Y -48.8821,Z 179,A -17.8261,B 5.7109,C 0.2836,E1 5.8677,E2 470.1069} C_DIS
LIN {X 128.882,Y -43.3793,Z 179,A -15.38,B 5.7112,C 0.2772,E1 5.8699,E2 467.661} C_DIS
LIN {X 129.8746,Y -40.3116,Z 179,A -14.0548,B 5.7113,C 0.274,E1 5.871,E2 466.3389} C_DIS
LIN {X 130.9205,Y -36.7695,Z 179,A -12.8278,B 5.7113,C 0.2749,E1 5.872,E2 465.1524} C_DIS
LIN {X 132.0316,Y -32.5626,Z 179,A -10.7028,B 5.7117,C 0.2652,E1 5.8735,E2 462.9888} C_DIS
LIN {X 132.8985,Y -28.8128,Z 179,A -9.2807,B 5.7118,C 0.2638,E1 5.8743,E2 461.5906} C_DIS
LIN {X 133.6108,Y -25.306,Z 179,A -7.7234,B 5.712,C 0.2588,E1 5.8752,E2 460.0257} C_DIS
LIN {X 134.5645,Y -19.615,Z 179,A -5.3374,B 5.7123,C 0.2526,E1 5.8762,E2 457.6435} C_DIS
LIN {X 135.0199,Y -16.1816,Z 179,A -3.9251,B 5.7125,C 0.2492,E1 5.8767,E2 456.236} C_DIS
LIN {X 135.4274,Y -12.3324,Z 179,A -2.3816,B 5.7125,C 0.246,E1 5.8771,E2 454.7023} C_DIS
LIN {X 135.7347,Y -8.2657,Z 179,A -0.1349,B 5.7132,C 0.2327,E1 5.8775,E2 452.3869} C_DIS
LIN {X 135.9433,Y -3.4316,Z 179,A 1.3868,B 5.7131,C 0.2351,E1 5.8777,E2 450.9295} C_DIS
LIN {X 135.9861,Y 0.5652,Z 179,A 3.1766,B 5.7133,C 0.2286,E1 5.8777,E2 449.125} C_DIS
LIN {X 135.8694,Y 5.6457,Z 179,A 5.5915,B 5.7137,C 0.2182,E1 5.8774,E2 446.6736} C_DIS
LIN {X 135.5782,Y 10.5451,Z 179,A 7.1456,B 5.7137,C 0.2204,E1 5.8771,E2 445.1833} C_DIS
LIN {X 135.2125,Y 14.4847,Z 179,A 8.6686,B 5.7137,C 0.2179,E1 5.8767,E2 443.6772} C_DIS
LIN {X 134.7202,Y 18.5251,Z 179,A 10.4121,B 5.7139,C 0.2126,E1 5.876,E2 441.929} C_DIS
LIN {X 134.1319,Y 22.379,Z 179,A 11.9617,B 5.714,C 0.2094,E1 5.8754,E2 440.3898} C_DIS
LIN {X 133.405,Y 26.3789,Z 179,A 13.7305,B 5.7143,C 0.2038,E1 5.8744,E2 438.613} C_DIS
LIN {X 132.6436,Y 29.9658,Z 179,A 15.1269,B 5.7143,C 0.2018,E1 5.8736,E2 437.2341} C_DIS
LIN {X 131.8354,Y 33.3405,Z 179,A 16.535,B 5.7144,C 0.1986,E1 5.8727,E2 435.8319} C_DIS
LIN {X 130.9339,Y 36.7214,Z 179,A 17.9485,B 5.7145,C 0.1955,E1 5.8716,E2 434.4251} C_DIS
LIN {X 129.7467,Y 40.7235,Z 179,A 19.7466,B 5.7147,C 0.1901,E1 5.8702,E2 432.6211} C_DIS
LIN {X 128.6341,Y 44.1089,Z 179,A 21.1838,B 5.7148,C 0.187,E1 5.8689,E2 431.191} C_DIS
LIN {X 127.4164,Y 47.5103,Z 179,A 22.6558,B 5.7149,C 0.1837,E1 5.8675,E2 429.7244} C_DIS
LIN {X 126.4291,Y 50.0844,Z 179,A 24.3762,B 5.7153,C 0.1721,E1 5.8657,E2 427.9333} C_DIS
LIN {X 124.5477,Y 54.5935,Z 179,A 25.8619,B 5.7152,C 0.1755,E1 5.8641,E2 426.5185} C_DIS
LIN {X 122.8515,Y 58.3072,Z 179,A 27.5138,B 5.7152,C 0.1721,E1 5.8621,E2 424.8742} C_DIS
LIN {X 121.3795,Y 61.3131,Z 179,A 28.9005,B 5.7154,C 0.1688,E1 5.8604,E2 423.4898} C_DIS
LIN {X 119.5818,Y 64.7534,Z 179,A 30.5792,B 5.7155,C 0.1641,E1 5.8582,E2 421.805} C_DIS
LIN {X 117.3834,Y 68.6574,Z 179,A 32.4101,B 5.7156,C 0.1603,E1 5.8557,E2 419.9803} C_DIS
LIN {X 115.1429,Y 72.3521,Z 179,A 34.2086,B 5.7157,C 0.1562,E1 5.853,E2 418.1838} C_DIS
LIN {X 112.5954,Y 76.2556,Z 179,A 36.0706,B 5.7158,C 0.1531,E1 5.8502,E2 416.3338} C_DIS
LIN {X 110.1575,Y 79.7369,Z 179,A 37.8503,B 5.7159,C 0.1491,E1 5.8473,E2 414.5548} C_DIS
LIN {X 108.0192,Y 82.6105,Z 179,A 39.2724,B 5.7159,C 0.1469,E1 5.8449,E2 413.143} C_DIS
LIN {X 105.5181,Y 85.7828,Z 179,A 40.8293,B 5.716,C 0.1453,E1 5.8422,E2 411.6034} C_DIS
LIN {X 103.3802,Y 88.3475,Z 179,A 42.3999,B 5.7162,C 0.1398,E1 5.8393,E2 410.0121} C_DIS
LIN {X 100.4035,Y 91.7167,Z 179,A 44.1058,B 5.7162,C 0.1385,E1 5.8362,E2 408.329} C_DIS
LIN {X 95.7692,Y 96.5449,Z 179,A 47.7576,B 5.7166,C 0.1206,E1 5.8288,E2 404.5731} C_DIS
LIN {X 91.2306,Y 100.8447,Z 179,A 49.5954,B 5.7165,C 0.1271,E1 5.8253,E2 402.8339} C_DIS
LIN {X 87.8675,Y 103.7883,Z 179,A 51.3418,B 5.7165,C 0.1255,E1 5.8216,E2 401.1042} C_DIS
LIN {X 84.8101,Y 106.301,Z 179,A 52.9435,B 5.7165,C 0.1234,E1 5.8181,E2 399.5103} C_DIS
LIN {X 81.9852,Y 108.4946,Z 179,A 54.5774,B 5.7166,C 0.119,E1 5.8145,E2 397.8606} C_DIS
LIN {X 78.3489,Y 111.149,Z 179,A 56.4214,B 5.7166,C 0.1165,E1 5.8103,E2 396.0229} C_DIS
LIN {X 74.6528,Y 113.6645,Z 179,A 58.3142,B 5.7168,C 0.1134,E1 5.8059,E2 394.129} C_DIS
LIN {X 70.8497,Y 116.0735,Z 179,A 60.1677,B 5.7168,C 0.1111,E1 5.8015,E2 392.2807} C_DIS
LIN {X 67.1178,Y 118.2706,Z 179,A 61.9852,B 5.7168,C 0.1086,E1 5.7971,E2 390.4641} C_DIS
LIN {X 63.4517,Y 120.2748,Z 179,A 63.6507,B 5.7168,C 0.1075,E1 5.7931,E2 388.8103} C_DIS
LIN {X 60.7192,Y 121.6785,Z 179,A 64.9943,B 5.7169,C 0.1051,E1 5.7897,E2 387.4608} C_DIS
LIN {X 57.2376,Y 123.3531,Z 179,A 66.4772,B 5.7169,C 0.1051,E1 5.786,E2 385.9957} C_DIS
LIN {X 54.2014,Y 124.7172,Z 179,A 67.917,B 5.7169,C 0.1029,E1 5.7823,E2 384.5514} C_DIS
LIN {X 51.0124,Y 126.0551,Z 179,A 69.1493,B 5.7169,C 0.1043,E1 5.7792,E2 383.3468} C_DIS
LIN {X 48.0716,Y 127.2061,Z 179,A 70.5212,B 5.7169,C 0.1023,E1 5.7756,E2 381.9701} C_DIS
LIN {X 44.7938,Y 128.3967,Z 179,A 72.1059,B 5.717,C 0.0993,E1 5.7714,E2 380.3716} C_DIS
LIN {X 42.1484,Y 129.2915,Z 179,A 73.2712,B 5.717,C 0.0984,E1 5.7683,E2 379.2079} C_DIS
LIN {X 35.879,Y 131.1695,Z 179,A 76.1877,B 5.7171,C 0.0941,E1 5.7605,E2 376.2726} C_DIS
LIN {X 31.9905,Y 132.1695,Z 179,A 77.6893,B 5.7171,C 0.0953,E1 5.7564,E2 374.7946} C_DIS
LIN {X 28.7307,Y 132.9162,Z 179,A 79.1105,B 5.7171,C 0.0942,E1 5.7526,E2 373.3723} C_DIS
LIN {X 25.6921,Y 133.5369,Z 179,A 80.4061,B 5.7171,C 0.0936,E1 5.749,E2 372.0784} C_DIS
LIN {X 22.3099,Y 134.1434,Z 179,A 81.8363,B 5.7171,C 0.0931,E1 5.7451,E2 370.6508} C_DIS
LIN {X 18.8263,Y 134.6772,Z 179,A 83.3373,B 5.7171,C 0.0922,E1 5.7409,E2 369.1483} C_DIS
LIN {X 14.2056,Y 135.2425,Z 179,A 85.7265,B 5.7172,C 0.0861,E1 5.7342,E2 366.7074} C_DIS
LIN {X 10.1575,Y 135.6065,Z 179,A 86.9665,B 5.7172,C 0.0916,E1 5.7309,E2 365.5259} C_DIS
LIN {X 6.778,Y 135.8172,Z 179,A 88.2281,B 5.7172,C 0.0934,E1 5.7274,E2 364.2849} C_DIS
LIN {X 3.435,Y 135.9432,Z 179,A 89.916,B 5.7172,C 0.0898,E1 5.7226,E2 362.5638} C_DIS
LIN {X -3.585,Y 135.9391,Z 179,A 92.8035,B 5.7172,C 0.0906,E1 5.7146,E2 359.6863} C_DIS
LIN {X -7.4834,Y 135.7817,Z 179,A 94.5398,B 5.7172,C 0.0897,E1 5.7097,E2 357.9395} C_DIS
LIN {X -11.7196,Y 135.4804,Z 179,A 96.5032,B 5.7172,C 0.0879,E1 5.7042,E2 355.9558} C_DIS
LIN {X -14.9357,Y 135.1639,Z 179,A 97.714,B 5.7172,C 0.0901,E1 5.7009,E2 354.764} C_DIS
LIN {X -19.0786,Y 134.6411,Z 179,A 99.4205,B 5.7172,C 0.0913,E1 5.6962,E2 353.0649} C_DIS
LIN {X -23.5178,Y 133.9376,Z 179,A 101.1956,B 5.7172,C 0.0935,E1 5.6913,E2 351.3054} C_DIS
LIN {X -26.9522,Y 133.2883,Z 179,A 102.738,B 5.7172,C 0.0935,E1 5.6871,E2 349.7553} C_DIS
LIN {X -30.342,Y 132.5577,Z 179,A 104.1395,B 5.7171,C 0.095,E1 5.6833,E2 348.3619} C_DIS
LIN {X -33.2775,Y 131.8514,Z 179,A 105.478,B 5.7171,C 0.0951,E1 5.6796,E2 347.0161} C_DIS
LIN {X -36.5046,Y 130.9946,Z 179,A 107.1087,B 5.7171,C 0.0936,E1 5.6751,E2 345.3591} C_DIS
LIN {X -41.0355,Y 129.647,Z 179,A 108.926,B 5.7171,C 0.0972,E1 5.6704,E2 343.5643} C_DIS
LIN {X -47.7399,Y 127.3303,Z 179,A 112.1047,B 5.7171,C 0.0978,E1 5.6619,E2 340.3645} C_DIS
LIN {X -52.1542,Y 125.5871,Z 179,A 114.064,B 5.717,C 0.1003,E1 5.6569,E2 338.4115} C_DIS
LIN {X -56.643,Y 123.628,Z 179,A 116.0272,B 5.717,C 0.1038,E1 5.6519,E2 336.4621} C_DIS
LIN {X -59.7401,Y 122.1615,Z 179,A 117.3317,B 5.7169,C 0.1071,E1 5.6487,E2 335.1756} C_DIS
LIN {X -62.7646,Y 120.6356,Z 179,A 118.9722,B 5.7169,C 0.1066,E1 5.6445,E2 333.5102} C_DIS
LIN {X -66.5504,Y 118.5905,Z 179,A 120.8402,B 5.7169,C 0.1084,E1 5.6399,E2 331.6369} C_DIS
LIN {X -69.9142,Y 116.6394,Z 179,A 123.275,B 5.7169,C 0.1023,E1 5.6339,E2 329.1055} C_DIS
LIN {X -75.1755,Y 113.3201,Z 179,A 125.1854,B 5.7167,C 0.1139,E1 5.6296,E2 327.2847} C_DIS
LIN {X -78.8295,Y 110.8091,Z 179,A 127.1002,B 5.7167,C 0.1164,E1 5.6252,E2 325.3657} C_DIS
LIN {X -82.4719,Y 108.1252,Z 179,A 129.0057,B 5.7167,C 0.1197,E1 5.621,E2 323.4619} C_DIS
LIN {X -85.9964,Y 105.3436,Z 179,A 130.9005,B 5.7166,C 0.123,E1 5.6169,E2 321.5682} C_DIS
LIN {X -89.2459,Y 102.6053,Z 179,A 132.765,B 5.7165,C 0.1255,E1 5.6129,E2 319.6961} C_DIS
LIN {X -92.7446,Y 99.4539,Z 179,A 134.7494,B 5.7165,C 0.1293,E1 5.6088,E2 317.7134} C_DIS
LIN {X -96.0511,Y 96.2648,Z 179,A 136.7377,B 5.7163,C 0.1326,E1 5.6048,E2 315.7202} C_DIS
LIN {X -99.1759,Y 93.0426,Z 179,A 138.6948,B 5.7163,C 0.1359,E1 5.601,E2 313.7567} C_DIS
LIN {X -102.1999,Y 89.7105,Z 179,A 140.6183,B 5.7162,C 0.1396,E1 5.5975,E2 311.8315} C_DIS
LIN {X -105.1041,Y 86.2894,Z 179,A 142.5562,B 5.7161,C 0.1433,E1 5.594,E2 309.8894} C_DIS
LIN {X -107.9657,Y 82.6804,Z 179,A 144.4575,B 5.716,C 0.148,E1 5.5907,E2 307.9946} C_DIS
LIN {X -110.4544,Y 79.3256,Z 179,A 146.33,B 5.7159,C 0.151,E1 5.5876,E2 306.1099} C_DIS
LIN {X -112.9866,Y 75.675,Z 179,A 148.7394,B 5.7159,C 0.1502,E1 5.5838,E2 303.6358} C_DIS
LIN {X -115.686,Y 71.4812,Z 179,A 150.1017,B 5.7156,C 0.1624,E1 5.5819,E2 302.3665} C_DIS
LIN {X -118.3209,Y 67.0295,Z 179,A 152.497,B 5.7155,C 0.1657,E1 5.5785,E2 299.9467} C_DIS
LIN {X -119.5799,Y 64.7561,Z 179,A 154.2711,B 5.7155,C 0.162,E1 5.5761,E2 298.0897} C_DIS
LIN {X -121.885,Y 60.3006,Z 179,A 155.739,B 5.7152,C 0.1735,E1 5.5743,E2 296.7035} C_DIS
LIN {X -123.3599,Y 57.2229,Z 179,A 157.2887,B 5.7152,C 0.1762,E1 5.5724,E2 295.1413} C_DIS
LIN {X -124.7951,Y 54.0212,Z 179,A 158.7541,B 5.715,C 0.1802,E1 5.5708,E2 293.6788} C_DIS
LIN {X -125.9147,Y 51.3607,Z 179,A 160.0986,B 5.715,C 0.1822,E1 5.5693,E2 292.3196} C_DIS
LIN {X -127.4802,Y 47.3399,Z 179,A 162.173,B 5.715,C 0.1846,E1 5.5673,E2 290.215} C_DIS
LIN {X -128.5813,Y 44.2614,Z 179,A 163.5298,B 5.7148,C 0.1886,E1 5.566,E2 288.862} C_DIS
LIN {X -129.9819,Y 39.9608,Z 179,A 165.1334,B 5.7145,C 0.1966,E1 5.5647,E2 287.2975} C_DIS
LIN {X -130.8742,Y 36.9348,Z 179,A 166.8116,B 5.7145,C 0.197,E1 5.5634,E2 285.5772} C_DIS
LIN {X -132.1476,Y 32.0815,Z 179,A 168.7779,B 5.7142,C 0.2042,E1 5.5621,E2 283.6311} C_DIS
LIN {X -132.9278,Y 28.6769,Z 179,A 170.304,B 5.7142,C 0.2078,E1 5.5611,E2 282.0995} C_DIS
LIN {X -133.7455,Y 24.5915,Z 179,A 172.0948,B 5.7139,C 0.2124,E1 5.5602,E2 280.3058} C_DIS
LIN {X -134.355,Y 20.9991,Z 179,A 173.6874,B 5.7138,C 0.2162,E1 5.5595,E2 278.7073} C_DIS
LIN {X -134.8895,Y 17.2397,Z 179,A 175.3849,B 5.7137,C 0.2198,E1 5.5588,E2 276.999} C_DIS
LIN {X -135.3479,Y 13.1599,Z 179,A 177.0938,B 5.7135,C 0.2249,E1 5.5583,E2 275.2941} C_DIS
LIN {X -135.6588,Y 9.4403,Z 179,A 178.794,B 5.7133,C 0.2282,E1 5.558,E2 273.5793} C_DIS
LIN {X -135.8842,Y 5.2669,Z 179,A -179.5031,B 5.7131,C 0.2338,E1 5.5578,E2 271.885} C_DIS
LIN {X -135.9824,Y 1.1533,Z 179,A -177.8095,B 5.7129,C 0.2391,E1 5.5577,E2 270.1978} C_DIS
LIN {X -135.9668,Y -2.3014,Z 179,A -176.2077,B 5.7128,C 0.2419,E1 5.5577,E2 268.5789} C_DIS
LIN {X -135.8335,Y -6.4529,Z 179,A -174.4286,B 5.7126,C 0.2466,E1 5.5579,E2 266.7975} C_DIS
LIN {X -135.6288,Y -9.8515,Z 179,A -172.9713,B 5.7124,C 0.2505,E1 5.5582,E2 265.3383} C_DIS
LIN {X -135.2923,Y -13.7391,Z 179,A -171.1426,B 5.7123,C 0.2534,E1 5.5587,E2 263.4878} C_DIS
LIN {X -134.8231,Y -17.7463,Z 179,A -169.5417,B 5.712,C 0.2591,E1 5.5592,E2 261.9005} C_DIS
LIN {X -134.2927,Y -21.4015,Z 179,A -167.8209,B 5.7119,C 0.262,E1 5.56,E2 260.1601} C_DIS
LIN {X -133.6158,Y -25.2799,Z 179,A -166.3592,B 5.7116,C 0.2684,E1 5.5607,E2 258.7242} C_DIS
LIN {X -132.9671,Y -28.4948,Z 179,A -164.861,B 5.7115,C 0.2712,E1 5.5615,E2 257.2124} C_DIS
LIN {X -132.3811,Y -31.1129,Z 179,A -163.3302,B 5.7115,C 0.2705,E1 5.5626,E2 255.632} C_DIS
LIN {X -131.5633,Y -34.404,Z 179,A -161.3344,B 5.7115,C 0.269,E1 5.5641,E2 253.565} C_DIS
LIN {X -129.8549,Y -40.3759,Z 179,A -159.3892,B 5.7109,C 0.2825,E1 5.5656,E2 251.7069} C_DIS
LIN {X -128.8538,Y -43.4637,Z 179,A -158.071,B 5.7107,C 0.2867,E1 5.5667,E2 250.3957} C_DIS
LIN {X -127.024,Y -48.5551,Z 179,A -155.6179,B 5.7105,C 0.2911,E1 5.5691,E2 247.922} C_DIS
LIN {X -125.5872,Y -52.154,Z 179,A -154.1128,B 5.7102,C 0.2966,E1 5.5707,E2 246.4339} C_DIS
LIN {X -124.3354,Y -55.0732,Z 179,A -152.6705,B 5.7101,C 0.299,E1 5.5723,E2 244.9791} C_DIS
LIN {X -122.3379,Y -59.382,Z 179,A -150.5741,B 5.7099,C 0.3032,E1 5.5748,E2 242.8718} C_DIS
LIN {X -120.5343,Y -62.9576,Z 179,A -149.0541,B 5.7095,C 0.309,E1 5.5767,E2 241.3736} C_DIS
LIN {X -117.3937,Y -68.6398,Z 179,A -146.0433,B 5.7093,C 0.313,E1 5.5809,E2 238.3294} C_DIS
LIN {X -114.9877,Y -72.5981,Z 179,A -144.0937,B 5.7091,C 0.3176,E1 5.5838,E2 236.3809} C_DIS
LIN {X -112.5771,Y -76.2827,Z 179,A -142.214,B 5.7088,C 0.3217,E1 5.5867,E2 234.4988} C_DIS
LIN {X -110.0025,Y -79.9507,Z 179,A -140.3276,B 5.7086,C 0.326,E1 5.5897,E2 232.6134} C_DIS
LIN {X -107.3171,Y -83.5209,Z 179,A -138.3363,B 5.7084,C 0.329,E1 5.5931,E2 230.6088} C_DIS
LIN {X -104.4883,Y -87.0345,Z 179,A -136.4049,B 5.7082,C 0.3328,E1 5.5966,E2 228.6741} C_DIS
LIN {X -101.8402,Y -90.1178,Z 179,A -134.7607,B 5.708,C 0.3371,E1 5.5996,E2 227.039} C_DIS
LIN {X -98.5911,Y -93.6622,Z 179,A -132.5765,B 5.7078,C 0.3395,E1 5.6038,E2 224.8352} C_DIS
LIN {X -95.6016,Y -96.7114,Z 179,A -130.7478,B 5.7076,C 0.3427,E1 5.6074,E2 223.0031} C_DIS
LIN {X -92.4057,Y -99.7695,Z 179,A -128.8538,B 5.7074,C 0.3459,E1 5.6112,E2 221.1055} C_DIS
LIN {X -89.0994,Y -102.7331,Z 179,A -126.9097,B 5.7073,C 0.3485,E1 5.6153,E2 219.1524} C_DIS
LIN {X -85.5692,Y -105.6911,Z 179,A -124.966,B 5.7071,C 0.3518,E1 5.6195,E2 217.2086} C_DIS
LIN {X -81.9423,Y -108.527,Z 179,A -123.0208,B 5.7069,C 0.3549,E1 5.6238,E2 215.2629} C_DIS
LIN {X -78.1939,Y -111.2583,Z 179,A -121.0367,B 5.7067,C 0.3577,E1 5.6283,E2 213.2751} C_DIS
LIN {X -74.6933,Y -113.6378,Z 179,A -119.2849,B 5.7065,C 0.3607,E1 5.6324,E2 211.5274} C_DIS
LIN {X -71.1128,Y -115.9121,Z 179,A -117.4438,B 5.7065,C 0.3626,E1 5.6368,E2 209.6794} C_DIS
LIN {X -67.1888,Y -118.2301,Z 179,A -115.4986,B 5.7063,C 0.3649,E1 5.6415,E2 207.7311} C_DIS
LIN {X -63.5614,Y -120.2172,Z 179,A -113.7805,B 5.7061,C 0.3673,E1 5.6457,E2 206.0159} C_DIS
LIN {X -60.7213,Y -121.6775,Z 179,A -112.3702,B 5.7061,C 0.3682,E1 5.6492,E2 204.5973} C_DIS
LIN {X -57.3273,Y -123.3116,Z 179,A -110.8687,B 5.7059,C 0.3709,E1 5.653,E2 203.1066} C_DIS
LIN {X -54.1571,Y -124.7363,Z 179,A -109.4119,B 5.7058,C 0.3726,E1 5.6567,E2 201.6506} C_DIS
LIN {X -51.2774,Y -125.9482,Z 179,A -108.1318,B 5.7057,C 0.3743,E1 5.66,E2 200.375} C_DIS
LIN {X -47.8275,Y -127.2976,Z 179,A -106.5003,B 5.7057,C 0.3749,E1 5.6643,E2 198.7342} C_DIS
LIN {X -43.7331,Y -128.764,Z 179,A -104.0237,B 5.706,C 0.3687,E1 5.6711,E2 196.1739} C_DIS
LIN {X -39.0745,Y -130.2532,Z 179,A -102.3885,B 5.7056,C 0.3753,E1 5.6753,E2 194.5936} C_DIS
LIN {X -35.0364,Y -131.3948,Z 179,A -100.7738,B 5.7054,C 0.3783,E1 5.6796,E2 192.9981} C_DIS
LIN {X -31.7305,Y -132.2322,Z 179,A -99.3282,B 5.7054,C 0.379,E1 5.6835,E2 191.551} C_DIS
LIN {X -27.8675,Y -133.1021,Z 179,A -97.5314,B 5.7054,C 0.3782,E1 5.6885,E2 189.7372} C_DIS
LIN {X -24.0274,Y -133.8465,Z 179,A -95.9938,B 5.7053,C 0.3802,E1 5.6926,E2 188.2133} C_DIS
LIN {X -20.9439,Y -134.3635,Z 179,A -94.7035,B 5.7053,C 0.381,E1 5.6962,E2 186.926} C_DIS
LIN {X -16.477,Y -134.9846,Z 179,A -92.3778,B 5.7055,C 0.3761,E1 5.7028,E2 184.5446} C_DIS
LIN {X -12.6928,Y -135.3928,Z 179,A -91.0839,B 5.7053,C 0.3803,E1 5.7063,E2 183.2903} C_DIS
LIN {X -6.1001,Y -135.8511,Z 179,A -88.4314,B 5.7051,C 0.3821,E1 5.7136,E2 180.6537} C_DIS
LIN {X 0.9634,Y -135.9823,Z 179,A -86.8663,B 5.7039,C 0.4,E1 5.7176,E2 179.2676} C_DIS
Enddeposition()
LIN {X 0.9634,Y -135.9823,Z 179,A -86.8667,B 5.7039,C 0.4,E1 5.7176,E2 179.2681} C_DIS
Startdeposition()
$VEL.CP = VEL_PRINT
LIN {X -0.9482,Y -136.8864,Z 179,A -86.8586,B 5.6699,C 0.3927,E1 5.6832,E2 179.2009} C_DIS
LIN {X -5.4536,Y -136.7809,Z 179,A -88.8499,B 5.6698,C 0.394,E1 5.6776,E2 181.2065} C_DIS
LIN {X -12.627,Y -136.3066,Z 179,A -91.5443,B 5.6701,C 0.3898,E1 5.6702,E2 183.8617} C_DIS
LIN {X -19.0056,Y -135.564,Z 179,A -94.8214,B 5.6696,C 0.3965,E1 5.6609,E2 187.2154} C_DIS
LIN {X -23.0396,Y -134.9375,Z 179,A -96.0717,B 5.67,C 0.3903,E1 5.6576,E2 188.4076} C_DIS
LIN {X -26.8594,Y -134.2291,Z 179,A -97.8378,B 5.67,C 0.3913,E1 5.6527,E2 190.1922} C_DIS
LIN {X -31.2494,Y -133.277,Z 179,A -99.6048,B 5.6701,C 0.389,E1 5.6479,E2 191.9452} C_DIS
LIN {X -34.7113,Y -132.4164,Z 179,A -101.1746,B 5.6701,C 0.389,E1 5.6437,E2 193.5253} C_DIS
LIN {X -38.6631,Y -131.3158,Z 179,A -102.8927,B 5.6701,C 0.3879,E1 5.639,E2 195.2439} C_DIS
LIN {X -43.5363,Y -129.7818,Z 179,A -105.0719,B 5.6703,C 0.3868,E1 5.6332,E2 197.4287} C_DIS
LIN {X -46.9415,Y -128.5901,Z 179,A -106.5114,B 5.6704,C 0.3847,E1 5.6295,E2 198.8595} C_DIS
LIN {X -50.672,Y -127.1662,Z 179,A -108.0969,B 5.6706,C 0.3822,E1 5.6254,E2 200.4343} C_DIS
LIN {X -53.2198,Y -126.121,Z 179,A -109.3402,B 5.6706,C 0.3821,E1 5.6221,E2 201.6893} C_DIS
LIN {X -56.1438,Y -124.8461,Z 179,A -110.7166,B 5.6706,C 0.3812,E1 5.6186,E2 203.0711} C_DIS
LIN {X -59.1816,Y -123.4348,Z 179,A -112.1461,B 5.6707,C 0.3799,E1 5.615,E2 204.5043} C_DIS
LIN {X -62.8782,Y -121.5963,Z 179,A -113.8844,B 5.6709,C 0.378,E1 5.6106,E2 206.244} C_DIS
LIN {X -65.5646,Y -120.1683,Z 179,A -115.2639,B 5.6709,C 0.3776,E1 5.6072,E2 207.6372} C_DIS
LIN {X -69.6172,Y -117.8673,Z 179,A -117.2347,B 5.671,C 0.3752,E1 5.6025,E2 209.6107} C_DIS
LIN {X -73.1887,Y -115.6831,Z 179,A -118.9969,B 5.6712,C 0.3729,E1 5.5983,E2 211.374} C_DIS
LIN {X -76.9148,Y -113.24,Z 179,A -120.8936,B 5.6713,C 0.3704,E1 5.5939,E2 213.2748} C_DIS
LIN {X -80.3958,Y -110.7956,Z 179,A -122.679,B 5.6715,C 0.3677,E1 5.5898,E2 215.0607} C_DIS
LIN {X -83.9885,Y -108.0976,Z 179,A -124.6239,B 5.6717,C 0.3653,E1 5.5855,E2 217.0135} C_DIS
LIN {X -87.5979,Y -105.1945,Z 179,A -126.6957,B 5.6718,C 0.3634,E1 5.5809,E2 219.102} C_DIS
LIN {X -91.3387,Y -101.9626,Z 179,A -128.6973,B 5.6721,C 0.3589,E1 5.5768,E2 221.0947} C_DIS
LIN {X -94.6097,Y -98.9351,Z 179,A -130.5683,B 5.6723,C 0.3555,E1 5.573,E2 222.966} C_DIS
LIN {X -97.9287,Y -95.6514,Z 179,A -132.5835,B 5.6725,C 0.3523,E1 5.569,E2 224.9886} C_DIS
LIN {X -102.6858,Y -90.5251,Z 179,A -135.3007,B 5.673,C 0.3442,E1 5.5639,E2 227.6783} C_DIS
LIN {X -104.6459,Y -88.2524,Z 179,A -136.8767,B 5.673,C 0.3449,E1 5.561,E2 229.2946} C_DIS
LIN {X -107.5447,Y -84.6954,Z 179,A -138.8103,B 5.6732,C 0.3408,E1 5.5576,E2 231.2293} C_DIS
LIN {X -110.355,Y -80.9995,Z 179,A -140.7262,B 5.6735,C 0.3362,E1 5.5544,E2 233.141} C_DIS
LIN {X -112.6894,Y -77.7196,Z 179,A -142.4996,B 5.6736,C 0.3333,E1 5.5515,E2 234.9249} C_DIS
LIN {X -114.9523,Y -74.3315,Z 179,A -144.2542,B 5.6738,C 0.3298,E1 5.5488,E2 236.6851} C_DIS
LIN {X -117.2816,Y -70.5991,Z 179,A -146.1083,B 5.6741,C 0.3255,E1 5.5461,E2 238.5401} C_DIS
LIN {X -119.7326,Y -66.3569,Z 179,A -148.1255,B 5.6744,C 0.3202,E1 5.5433,E2 240.552} C_DIS
LIN {X -121.7396,Y -62.5968,Z 179,A -150.0164,B 5.6746,C 0.3168,E1 5.5409,E2 242.4556} C_DIS
LIN {X -123.641,Y -58.7502,Z 179,A -151.8351,B 5.6748,C 0.3125,E1 5.5386,E2 244.2762} C_DIS
LIN {X -125.0414,Y -55.707,Z 179,A -153.2287,B 5.675,C 0.3088,E1 5.537,E2 245.668} C_DIS
LIN {X -126.4136,Y -52.5193,Z 179,A -154.7299,B 5.6752,C 0.3055,E1 5.5354,E2 247.1745} C_DIS
LIN {X -127.6155,Y -49.5268,Z 179,A -156.0433,B 5.6754,C 0.3016,E1 5.5341,E2 248.4826} C_DIS
LIN {X -129.6582,Y -43.9075,Z 179,A -158.5977,B 5.6757,C 0.2955,E1 5.5317,E2 251.0422} C_DIS
LIN {X -130.5991,Y -41.0236,Z 179,A -160.0136,B 5.6758,C 0.2934,E1 5.5304,E2 252.4757} C_DIS
LIN {X -132.7168,Y -33.5398,Z 179,A -163.2922,B 5.6763,C 0.2848,E1 5.528,E2 255.7552} C_DIS
LIN {X -133.3339,Y -31.0003,Z 179,A -164.4953,B 5.6763,C 0.2828,E1 5.5272,E2 256.9714} C_DIS
LIN {X -134.1792,Y -27.1043,Z 179,A -166.0902,B 5.6766,C 0.2774,E1 5.5263,E2 258.5559} C_DIS
LIN {X -134.7807,Y -23.935,Z 179,A -167.5205,B 5.6768,C 0.2744,E1 5.5256,E2 259.9952} C_DIS
LIN {X -135.422,Y -19.9993,Z 179,A -169.3846,B 5.6769,C 0.2715,E1 5.5248,E2 261.8826} C_DIS
LIN {X -135.9886,Y -15.6875,Z 179,A -171.2287,B 5.6772,C 0.2666,E1 5.5241,E2 263.7283} C_DIS
LIN {X -136.3894,Y -11.6908,Z 179,A -172.8316,B 5.6774,C 0.2611,E1 5.5237,E2 265.3202} C_DIS
LIN {X -136.6475,Y -8.1399,Z 179,A -174.4344,B 5.6776,C 0.2579,E1 5.5234,E2 266.936} C_DIS
LIN {X -136.8307,Y -4.0174,Z 179,A -176.1503,B 5.6778,C 0.2529,E1 5.5232,E2 268.6492} C_DIS
LIN {X -136.8925,Y 0.0485,Z 179,A -178.0301,B 5.6779,C 0.2497,E1 5.5232,E2 270.5499} C_DIS
LIN {X -136.8286,Y 4.0934,Z 179,A -179.7268,B 5.6781,C 0.2449,E1 5.5233,E2 272.2456} C_DIS
LIN {X -136.6355,Y 8.3357,Z 179,A 178.592,B 5.6784,C 0.2389,E1 5.5236,E2 273.9134} C_DIS
LIN {X -136.3827,Y 11.77,Z 179,A 177.1632,B 5.6786,C 0.2347,E1 5.5239,E2 275.3395} C_DIS
LIN {X -136.1141,Y 14.5486,Z 179,A 175.8847,B 5.6786,C 0.2324,E1 5.5242,E2 276.6307} C_DIS
LIN {X -135.7036,Y 17.9801,Z 179,A 174.4494,B 5.6788,C 0.2282,E1 5.5247,E2 278.0634} C_DIS
LIN {X -135.2572,Y 21.0757,Z 179,A 173.0448,B 5.6789,C 0.2254,E1 5.5253,E2 279.4787} C_DIS
LIN {X -134.542,Y 25.2455,Z 179,A 171.1719,B 5.6791,C 0.2213,E1 5.5262,E2 281.3629} C_DIS
LIN {X -133.8206,Y 28.8219,Z 179,A 169.6851,B 5.6793,C 0.2167,E1 5.5271,E2 282.8434} C_DIS
LIN {X -133.043,Y 32.2215,Z 179,A 168.1071,B 5.6793,C 0.2137,E1 5.5281,E2 284.4347} C_DIS
LIN {X -132.1,Y 35.8979,Z 179,A 165.9743,B 5.6793,C 0.2143,E1 5.5297,E2 286.633} C_DIS
LIN {X -130.804,Y 40.3613,Z 179,A 164.5172,B 5.6797,C 0.2045,E1 5.5308,E2 288.0286} C_DIS
LIN {X -128.3319,Y 47.6412,Z 179,A 161.4323,B 5.6801,C 0.1946,E1 5.5336,E2 291.0943} C_DIS
LIN {X -126.6493,Y 51.9544,Z 179,A 159.2759,B 5.6801,C 0.1915,E1 5.5359,E2 293.276} C_DIS
LIN {X -125.532,Y 54.593,Z 179,A 158.0187,B 5.6803,C 0.1889,E1 5.5373,E2 294.5392} C_DIS
LIN {X -123.8637,Y 58.2839,Z 179,A 156.3271,B 5.6804,C 0.1845,E1 5.5392,E2 296.2288} C_DIS
LIN {X -122.6518,Y 60.7881,Z 179,A 154.7797,B 5.6804,C 0.1851,E1 5.5412,E2 297.822} C_DIS
LIN {X -121.0729,Y 63.8748,Z 179,A 153.6254,B 5.6806,C 0.1786,E1 5.5427,E2 298.9388} C_DIS
LIN {X -119.0917,Y 67.5015,Z 179,A 151.7484,B 5.6806,C 0.1757,E1 5.5452,E2 300.8324} C_DIS
LIN {X -116.8981,Y 71.2329,Z 179,A 149.7345,B 5.6808,C 0.1732,E1 5.5482,E2 302.8693} C_DIS
LIN {X -113.7996,Y 76.0842,Z 179,A 147.4553,B 5.681,C 0.1662,E1 5.5516,E2 305.1305} C_DIS
LIN {X -111.364,Y 79.6065,Z 179,A 145.6083,B 5.681,C 0.1625,E1 5.5546,E2 306.9826} C_DIS
LIN {X -108.6459,Y 83.278,Z 179,A 143.6938,B 5.6812,C 0.1582,E1 5.5578,E2 308.8957} C_DIS
LIN {X -105.8981,Y 86.7454,Z 179,A 141.7658,B 5.6812,C 0.1548,E1 5.5612,E2 310.8314} C_DIS
LIN {X -103.0423,Y 90.1191,Z 179,A 139.9115,B 5.6814,C 0.1509,E1 5.5645,E2 312.6846} C_DIS
LIN {X -100.0224,Y 93.4597,Z 179,A 137.9751,B 5.6814,C 0.1474,E1 5.5682,E2 314.6257} C_DIS
LIN {X -96.8979,Y 96.6955,Z 179,A 136.0587,B 5.6816,C 0.144,E1 5.572,E2 316.5446} C_DIS
LIN {X -93.6511,Y 99.8437,Z 179,A 134.0983,B 5.6816,C 0.1409,E1 5.5759,E2 318.5115} C_DIS
LIN {X -90.2946,Y 102.8891,Z 179,A 132.1626,B 5.6817,C 0.1377,E1 5.58,E2 320.4503} C_DIS
LIN {X -86.8551,Y 105.8084,Z 179,A 130.2574,B 5.6818,C 0.1345,E1 5.5841,E2 322.356} C_DIS
LIN {X -83.3581,Y 108.5846,Z 179,A 128.3531,B 5.6818,C 0.1316,E1 5.5883,E2 324.2631} C_DIS
LIN {X -79.7066,Y 111.2925,Z 179,A 126.4458,B 5.6819,C 0.1285,E1 5.5926,E2 326.1694} C_DIS
LIN {X -76.0746,Y 113.806,Z 179,A 124.5859,B 5.682,C 0.1256,E1 5.5969,E2 328.0293} C_DIS
LIN {X -71.5561,Y 116.6999,Z 179,A 122.4992,B 5.6821,C 0.1206,E1 5.6017,E2 330.0948} C_DIS
LIN {X -68.5081,Y 118.5149,Z 179,A 120.8248,B 5.6821,C 0.1205,E1 5.6058,E2 331.7911} C_DIS
LIN {X -64.5744,Y 120.7036,Z 179,A 118.9719,B 5.6821,C 0.1176,E1 5.6103,E2 333.6389} C_DIS
LIN {X -61.3661,Y 122.3659,Z 179,A 117.4503,B 5.6822,C 0.1158,E1 5.6141,E2 335.1605} C_DIS
LIN {X -58.7684,Y 123.6323,Z 179,A 116.2087,B 5.6822,C 0.1147,E1 5.6173,E2 336.4049} C_DIS
LIN {X -55.1806,Y 125.2769,Z 179,A 114.5692,B 5.6822,C 0.1126,E1 5.6214,E2 338.0418} C_DIS
LIN {X -50.7457,Y 127.1365,Z 179,A 112.4155,B 5.6822,C 0.112,E1 5.627,E2 340.2111} C_DIS
LIN {X -43.7752,Y 129.7022,Z 179,A 109.4982,B 5.6824,C 0.107,E1 5.6346,E2 343.1032} C_DIS
LIN {X -39.0897,Y 131.1909,Z 179,A 107.389,B 5.6824,C 0.1059,E1 5.6403,E2 345.2174} C_DIS
LIN {X -36.4477,Y 131.9485,Z 179,A 106.1929,B 5.6824,C 0.1056,E1 5.6435,E2 346.4183} C_DIS
LIN {X -33.5074,Y 132.725,Z 179,A 104.8604,B 5.6824,C 0.1054,E1 5.6471,E2 347.7572} C_DIS
LIN {X -29.507,Y 133.6727,Z 179,A 103.0476,B 5.6824,C 0.1054,E1 5.6521,E2 349.5801} C_DIS
LIN {X -25.5533,Y 134.4832,Z 179,A 101.3786,B 5.6824,C 0.1043,E1 5.6567,E2 351.2457} C_DIS
LIN {X -21.9614,Y 135.1174,Z 179,A 99.8079,B 5.6824,C 0.1041,E1 5.661,E2 352.8209} C_DIS
LIN {X -17.872,Y 135.7177,Z 179,A 98.136,B 5.6824,C 0.1028,E1 5.6656,E2 354.4848} C_DIS
LIN {X -14.3235,Y 136.1384,Z 179,A 96.3691,B 5.6824,C 0.1056,E1 5.6706,E2 356.2837} C_DIS
LIN {X -10.9265,Y 136.4537,Z 179,A 94.7936,B 5.6824,C 0.107,E1 5.675,E2 357.8763} C_DIS
LIN {X -6.8626,Y 136.7174,Z 179,A 93.6357,B 5.6825,C 0.1003,E1 5.6781,E2 358.9673} C_DIS
LIN {X -4.03,Y 136.8304,Z 179,A 91.4913,B 5.6823,C 0.1117,E1 5.6844,E2 361.2265} C_DIS
LIN {X 2.2886,Y 136.8704,Z 179,A 90.0325,B 5.6826,C 0.0976,E1 5.6881,E2 362.5412} C_DIS
LIN {X 8.1881,Y 136.6446,Z 179,A 87.4743,B 5.6826,C 0.099,E1 5.6952,E2 365.1092} C_DIS
LIN {X 11.4741,Y 136.4077,Z 179,A 84.8651,B 5.6822,C 0.1145,E1 5.7029,E2 367.8662} C_DIS
LIN {X 18.5969,Y 135.6224,Z 179,A 82.9063,B 5.6825,C 0.1028,E1 5.708,E2 369.6989} C_DIS
LIN {X 22.6885,Y 134.9961,Z 179,A 81.1759,B 5.6825,C 0.1036,E1 5.7127,E2 371.4284} C_DIS
LIN {X 25.904,Y 134.4161,Z 179,A 79.7271,B 5.6825,C 0.1054,E1 5.7167,E2 372.8867} C_DIS
LIN {X 29.426,Y 133.6902,Z 179,A 78.1706,B 5.6824,C 0.107,E1 5.721,E2 374.449} C_DIS
LIN {X 33.4074,Y 132.7504,Z 179,A 76.5124,B 5.6824,C 0.1075,E1 5.7255,E2 376.1002} C_DIS
LIN {X 37.5087,Y 131.6518,Z 179,A 74.5455,B 5.6824,C 0.1114,E1 5.7308,E2 378.0897} C_DIS
LIN {X 42.2352,Y 130.2121,Z 179,A 72.783,B 5.6824,C 0.1092,E1 5.7354,E2 379.8148} C_DIS
LIN {X 44.7262,Y 129.3762,Z 179,A 71.6343,B 5.6824,C 0.1109,E1 5.7385,E2 380.9692} C_DIS
LIN {X 48.8153,Y 127.8918,Z 179,A 69.8948,B 5.6823,C 0.1117,E1 5.743,E2 382.6986} C_DIS
LIN {X 51.4061,Y 126.8703,Z 179,A 68.7178,B 5.6823,C 0.1131,E1 5.7461,E2 383.8768} C_DIS
LIN {X 54.4601,Y 125.5895,Z 179,A 67.3435,B 5.6823,C 0.1145,E1 5.7496,E2 385.2495} C_DIS
LIN {X 57.6128,Y 124.1748,Z 179,A 65.9165,B 5.6823,C 0.116,E1 5.7532,E2 386.6739} C_DIS
LIN {X 61.2559,Y 122.421,Z 179,A 64.2554,B 5.6822,C 0.1178,E1 5.7574,E2 388.3312} C_DIS
LIN {X 64.5541,Y 120.7145,Z 179,A 62.6009,B 5.6822,C 0.1212,E1 5.7615,E2 389.9979} C_DIS
LIN {X 68.5887,Y 118.4683,Z 179,A 60.7183,B 5.6821,C 0.1233,E1 5.7661,E2 391.8744} C_DIS
LIN {X 72.4027,Y 116.1766,Z 179,A 58.881,B 5.6821,C 0.1258,E1 5.7704,E2 393.7087} C_DIS
LIN {X 76.2584,Y 113.6833,Z 179,A 56.992,B 5.6819,C 0.1284,E1 5.7748,E2 395.5937} C_DIS
LIN {X 79.6065,Y 111.364,Z 179,A 55.3408,B 5.6819,C 0.1304,E1 5.7786,E2 397.2385} C_DIS
LIN {X 82.9883,Y 108.8675,Z 179,A 53.5485,B 5.6819,C 0.1339,E1 5.7826,E2 399.035} C_DIS
LIN {X 85.91,Y 106.5768,Z 179,A 52.0044,B 5.6818,C 0.1366,E1 5.786,E2 400.5781} C_DIS
LIN {X 89.5144,Y 103.5681,Z 179,A 50.1434,B 5.6818,C 0.1387,E1 5.7899,E2 402.4267} C_DIS
LIN {X 92.6547,Y 100.7682,Z 179,A 48.1995,B 5.6816,C 0.1448,E1 5.794,E2 404.3933} C_DIS
LIN {X 94.9892,Y 98.5712,Z 179,A 47.345,B 5.6816,C 0.1404,E1 5.7956,E2 405.1882} C_DIS
LIN {X 98.5984,Y 94.9612,Z 179,A 44.8158,B 5.6814,C 0.1504,E1 5.8006,E2 407.7663} C_DIS
LIN {X 101.3968,Y 91.9664,Z 179,A 43.2784,B 5.6814,C 0.1515,E1 5.8035,E2 409.2822} C_DIS
LIN {X 104.4577,Y 88.4748,Z 179,A 41.3058,B 5.6813,C 0.1561,E1 5.8071,E2 411.2589} C_DIS
LIN {X 106.8331,Y 85.5921,Z 179,A 39.6849,B 5.6811,C 0.1604,E1 5.81,E2 412.8874} C_DIS
LIN {X 110.0391,Y 81.4291,Z 179,A 37.6821,B 5.6811,C 0.1625,E1 5.8133,E2 414.8667} C_DIS
LIN {X 112.4213,Y 78.1064,Z 179,A 36.0245,B 5.681,C 0.1657,E1 5.816,E2 416.5184} C_DIS
LIN {X 114.7081,Y 74.7077,Z 179,A 34.3099,B 5.6809,C 0.1698,E1 5.8186,E2 418.2336} C_DIS
LIN {X 117.1411,Y 70.8315,Z 179,A 32.4333,B 5.6807,C 0.1739,E1 5.8214,E2 420.1062} C_DIS
LIN {X 119.387,Y 66.9769,Z 179,A 30.6609,B 5.6807,C 0.1771,E1 5.8238,E2 421.8678} C_DIS
LIN {X 121.3457,Y 63.3554,Z 179,A 29.0188,B 5.6805,C 0.1802,E1 5.8259,E2 423.5005} C_DIS
LIN {X 122.9044,Y 60.2761,Z 179,A 27.5904,B 5.6805,C 0.1836,E1 5.8277,E2 424.9276} C_DIS
LIN {X 124.3998,Y 57.1262,Z 179,A 26.1221,B 5.6803,C 0.1875,E1 5.8295,E2 426.3977} C_DIS
LIN {X 126.4796,Y 52.3611,Z 179,A 24.0501,B 5.6802,C 0.1916,E1 5.8317,E2 428.458} C_DIS
LIN {X 127.6891,Y 49.3375,Z 179,A 22.792,B 5.6802,C 0.1937,E1 5.833,E2 429.7037} C_DIS
LIN {X 128.9191,Y 46.0289,Z 179,A 21.2964,B 5.68,C 0.1979,E1 5.8344,E2 431.2025} C_DIS
LIN {X 129.8858,Y 43.224,Z 179,A 20.0889,B 5.6799,C 0.2007,E1 5.8355,E2 432.4064} C_DIS
LIN {X 130.9461,Y 39.8973,Z 179,A 18.646,B 5.6797,C 0.2044,E1 5.8367,E2 433.8479} C_DIS
LIN {X 131.9488,Y 36.4466,Z 179,A 17.2107,B 5.6797,C 0.2075,E1 5.8378,E2 435.2755} C_DIS
LIN {X 132.7389,Y 33.4529,Z 179,A 15.8868,B 5.6795,C 0.2115,E1 5.8387,E2 436.6037} C_DIS
LIN {X 133.7385,Y 29.2022,Z 179,A 14.093,B 5.6793,C 0.216,E1 5.8398,E2 438.3945} C_DIS
LIN {X 134.4545,Y 25.7033,Z 179,A 12.6759,B 5.6792,C 0.219,E1 5.8406,E2 439.8028} C_DIS
LIN {X 135.0329,Y 22.468,Z 179,A 11.2768,B 5.679,C 0.2232,E1 5.8413,E2 441.2058} C_DIS
LIN {X 135.5692,Y 18.9694,Z 179,A 9.8045,B 5.6789,C 0.2273,E1 5.8419,E2 442.678} C_DIS
LIN {X 136.2327,Y 13.396,Z 179,A 7.7935,B 5.6789,C 0.2287,E1 5.8425,E2 444.6482} C_DIS
LIN {X 136.7993,Y 4.9804,Z 179,A 4.4397,B 5.6785,C 0.236,E1 5.8431,E2 447.9825} C_DIS
LIN {X 136.8841,Y -1.398,Z 179,A 1.3793,B 5.6779,C 0.2497,E1 5.8431,E2 451.0943} C_DIS
LIN {X 136.5547,Y -9.576,Z 179,A -2.308,B 5.6773,C 0.2635,E1 5.8426,E2 454.8171} C_DIS
LIN {X 136.1565,Y -14.1553,Z 179,A -3.5343,B 5.6775,C 0.2582,E1 5.8423,E2 455.9572} C_DIS
LIN {X 135.6545,Y -18.3545,Z 179,A -5.5349,B 5.6771,C 0.2668,E1 5.8416,E2 457.9884} C_DIS
LIN {X 134.87,Y -23.4349,Z 179,A -7.6929,B 5.6769,C 0.2729,E1 5.8406,E2 460.149} C_DIS
LIN {X 134.1455,Y -27.2699,Z 179,A -9.0868,B 5.6769,C 0.2738,E1 5.8399,E2 461.514} C_DIS
LIN {X 133.4063,Y -30.6833,Z 179,A -10.5365,B 5.6766,C 0.2777,E1 5.839,E2 462.9634} C_DIS
LIN {X 132.3786,Y -34.853,Z 179,A -12.3734,B 5.6764,C 0.2833,E1 5.8377,E2 464.8068} C_DIS
LIN {X 131.1459,Y -39.2435,Z 179,A -14.1165,B 5.6762,C 0.286,E1 5.8364,E2 466.5307} C_DIS
LIN {X 130.1478,Y -42.4364,Z 179,A -15.6576,B 5.6759,C 0.292,E1 5.8351,E2 468.0909} C_DIS
LIN {X 128.6923,Y -46.6579,Z 179,A -17.3338,B 5.6759,C 0.2941,E1 5.8335,E2 469.7442} C_DIS
LIN {X 127.2723,Y -50.4088,Z 179,A -18.9474,B 5.6756,C 0.2976,E1 5.8319,E2 471.3511} C_DIS
LIN {X 126.0378,Y -53.4191,Z 179,A -20.2682,B 5.6755,C 0.3006,E1 5.8305,E2 472.6679} C_DIS
LIN {X 124.9626,Y -55.8833,Z 179,A -21.4847,B 5.6752,C 0.305,E1 5.8291,E2 473.8969} C_DIS
LIN {X 123.0804,Y -59.9192,Z 179,A -23.2815,B 5.675,C 0.3088,E1 5.827,E2 475.6869} C_DIS
LIN {X 120.2944,Y -65.3334,Z 179,A -25.751,B 5.6747,C 0.3142,E1 5.8238,E2 478.1487} C_DIS
LIN {X 118.1995,Y -69.0516,Z 179,A -27.5558,B 5.6745,C 0.3189,E1 5.8213,E2 479.9575} C_DIS
LIN {X 115.9154,Y -72.8207,Z 179,A -29.3694,B 5.6742,C 0.323,E1 5.8186,E2 481.7688} C_DIS
LIN {X 113.403,Y -76.674,Z 179,A -31.2382,B 5.674,C 0.3268,E1 5.8157,E2 483.6321} C_DIS
LIN {X 110.9497,Y -80.1831,Z 179,A -32.9932,B 5.6738,C 0.3305,E1 5.8129,E2 485.384} C_DIS
LIN {X 108.3709,Y -83.6359,Z 179,A -34.7543,B 5.6736,C 0.3341,E1 5.8099,E2 487.1412} C_DIS
LIN {X 105.6015,Y -87.1064,Z 179,A -36.6001,B 5.6734,C 0.3381,E1 5.8067,E2 488.987} C_DIS
LIN {X 102.6442,Y -90.5722,Z 179,A -38.3968,B 5.6732,C 0.3407,E1 5.8034,E2 490.7713} C_DIS
LIN {X 98.7794,Y -94.7726,Z 179,A -40.545,B 5.6732,C 0.3422,E1 5.7994,E2 492.8908} C_DIS
LIN {X 97.0032,Y -96.5896,Z 179,A -41.9139,B 5.6727,C 0.349,E1 5.7966,E2 494.2998} C_DIS
LIN {X 91.8789,Y -101.4762,Z 179,A -45.0867,B 5.6721,C 0.3581,E1 5.7901,E2 497.5019} C_DIS
LIN {X 88.7786,Y -104.1994,Z 179,A -46.3859,B 5.6723,C 0.3551,E1 5.7874,E2 498.7479} C_DIS
LIN {X 85.5312,Y -106.8816,Z 179,A -48.1826,B 5.6721,C 0.359,E1 5.7835,E2 500.5504} C_DIS
LIN {X 82.0438,Y -109.5814,Z 179,A -50.0242,B 5.6719,C 0.3622,E1 5.7794,E2 502.393} C_DIS
LIN {X 78.3082,Y -112.2809,Z 179,A -51.9009,B 5.6717,C 0.3648,E1 5.7752,E2 504.2646} C_DIS
LIN {X 74.3989,Y -114.9086,Z 179,A -53.8012,B 5.6716,C 0.3671,E1 5.7708,E2 506.1574} C_DIS
LIN {X 70.7364,Y -117.1986,Z 179,A -55.5817,B 5.6714,C 0.3696,E1 5.7665,E2 507.9358} C_DIS
LIN {X 67.0893,Y -119.3238,Z 179,A -57.3213,B 5.6713,C 0.3719,E1 5.7623,E2 509.6734} C_DIS
LIN {X 63.4904,Y -121.2748,Z 179,A -59.0265,B 5.6711,C 0.3742,E1 5.7581,E2 511.3787} C_DIS
LIN {X 60.0991,Y -122.9917,Z 179,A -60.5391,B 5.6711,C 0.3753,E1 5.7544,E2 512.8825} C_DIS
LIN {X 54.7577,Y -125.4608,Z 179,A -62.8197,B 5.671,C 0.3759,E1 5.7486,E2 515.1414} C_DIS
LIN {X 46.1989,Y -128.8578,Z 179,A -66.8179,B 5.6706,C 0.3824,E1 5.7382,E2 519.1612} C_DIS
LIN {X 42.8754,Y -130.0018,Z 179,A -68.2079,B 5.6706,C 0.3827,E1 5.7345,E2 520.5418} C_DIS
LIN {X 39.4524,Y -131.0822,Z 179,A -69.697,B 5.6704,C 0.384,E1 5.7305,E2 522.0303} C_DIS
LIN {X 36.78,Y -131.8555,Z 179,A -70.8737,B 5.6704,C 0.3852,E1 5.7274,E2 523.2092} C_DIS
LIN {X 33.1901,Y -132.8056,Z 179,A -72.3703,B 5.6704,C 0.3857,E1 5.7233,E2 524.6994} C_DIS
LIN {X 30.249,Y -133.5055,Z 179,A -73.6561,B 5.6702,C 0.387,E1 5.7198,E2 525.9887} C_DIS
LIN {X 26.9674,Y -134.2071,Z 179,A -75.0147,B 5.6702,C 0.3873,E1 5.7161,E2 527.3422} C_DIS
LIN {X 24.0743,Y -134.7557,Z 179,A -76.2865,B 5.6702,C 0.3886,E1 5.7126,E2 528.6198} C_DIS
LIN {X 15.8896,Y -135.9644,Z 179,A -79.5181,B 5.6702,C 0.3874,E1 5.7038,E2 531.8237} C_DIS
LIN {X 8.9439,Y -136.598,Z 179,A -82.7831,B 5.6698,C 0.393,E1 5.6946,E2 535.135} C_DIS
LIN {X 1.8148,Y -136.8783,Z 179,A -85.5205,B 5.67,C 0.3905,E1 5.687,E2 537.8419} C_DIS
LIN {X 1.8148,Y -136.8783,Z 179,A -85.5205,B 5.67,C 0.3905,E1 5.687,E2 537.8419} C_DIS
Enddeposition()
LIN {X 0.9805,Y -137.7877,Z 179,A -85.4977,B 5.6362,C 0.3885,E1 5.6532,E2 537.8129} C_DIS
Startdeposition()
$VEL.CP = VEL_PRINT
LIN {X 4.993,Y -137.7029,Z 179,A -83.6752,B 5.6364,C 0.3862,E1 5.6584,E2 535.9696} C_DIS
LIN {X 7.6943,Y -137.58,Z 179,A -82.4345,B 5.6365,C 0.3843,E1 5.6619,E2 534.7131} C_DIS
LIN {X 10.8138,Y -137.37,Z 179,A -81.2531,B 5.6365,C 0.3855,E1 5.6651,E2 533.5467} C_DIS
LIN {X 14.5297,Y -137.0247,Z 179,A -79.6849,B 5.6365,C 0.3846,E1 5.6695,E2 531.9753} C_DIS
LIN {X 18.6981,Y -136.5205,Z 179,A -77.9627,B 5.6365,C 0.3841,E1 5.6743,E2 530.2554} C_DIS
LIN {X 21.8798,Y -136.0468,Z 179,A -76.6297,B 5.6365,C 0.3834,E1 5.678,E2 528.9222} C_DIS
LIN {X 25.4832,Y -135.4163,Z 179,A -75.1142,B 5.6366,C 0.3825,E1 5.6821,E2 527.4064} C_DIS
LIN {X 28.6874,Y -134.7738,Z 179,A -73.7293,B 5.6367,C 0.3812,E1 5.6859,E2 526.0172} C_DIS
LIN {X 31.891,Y -134.0519,Z 179,A -72.5558,B 5.6367,C 0.3828,E1 5.689,E2 524.8681} C_DIS
LIN {X 34.7007,Y -133.3541,Z 179,A -71.2071,B 5.6368,C 0.3798,E1 5.6928,E2 523.4996} C_DIS
LIN {X 37.9154,Y -132.476,Z 179,A -69.8304,B 5.6369,C 0.3787,E1 5.6965,E2 522.1232} C_DIS
LIN {X 41.5233,Y -131.3878,Z 179,A -68.27,B 5.6369,C 0.3773,E1 5.7006,E2 520.5625} C_DIS
LIN {X 44.745,Y -130.3258,Z 179,A -66.8751,B 5.6371,C 0.3761,E1 5.7043,E2 519.1687} C_DIS
LIN {X 47.9425,Y -129.1837,Z 179,A -65.4754,B 5.6371,C 0.3747,E1 5.708,E2 517.7696} C_DIS
LIN {X 51.1281,Y -127.9564,Z 179,A -64.0453,B 5.6373,C 0.3729,E1 5.7117,E2 516.3371} C_DIS
LIN {X 54.4338,Y -126.585,Z 179,A -62.6107,B 5.6373,C 0.3719,E1 5.7154,E2 514.9084} C_DIS
LIN {X 57.4498,Y -125.2455,Z 179,A -61.2371,B 5.6375,C 0.3701,E1 5.7189,E2 513.5336} C_DIS
LIN {X 60.5793,Y -123.762,Z 179,A -59.9744,B 5.6375,C 0.3707,E1 5.722,E2 512.2931} C_DIS
LIN {X 63.2885,Y -122.4011,Z 179,A -58.4381,B 5.6378,C 0.365,E1 5.7259,E2 510.7197} C_DIS
LIN {X 67.3282,Y -120.2258,Z 179,A -56.6822,B 5.6378,C 0.3644,E1 5.7302,E2 508.9823} C_DIS
LIN {X 70.7336,Y -118.2543,Z 179,A -54.9858,B 5.6381,C 0.361,E1 5.7343,E2 507.2767} C_DIS
LIN {X 74.5567,Y -115.8822,Z 179,A -53.1288,B 5.6382,C 0.3582,E1 5.7387,E2 505.42} C_DIS
LIN {X 78.3355,Y -113.3623,Z 179,A -51.3605,B 5.6383,C 0.3567,E1 5.7427,E2 503.6659} C_DIS
LIN {X 81.2234,Y -111.3114,Z 179,A -49.8553,B 5.6385,C 0.3537,E1 5.7461,E2 502.1553} C_DIS
LIN {X 84.2429,Y -109.0433,Z 179,A -48.2859,B 5.6387,C 0.3508,E1 5.7496,E2 500.5846} C_DIS
LIN {X 87.6756,Y -106.303,Z 179,A -46.5556,B 5.6388,C 0.3488,E1 5.7534,E2 498.8653} C_DIS
LIN {X 90.433,Y -103.9673,Z 179,A -45.0096,B 5.639,C 0.3453,E1 5.7566,E2 497.3123} C_DIS
LIN {X 93.5801,Y -101.1446,Z 179,A -43.3633,B 5.6392,C 0.3434,E1 5.76,E2 495.6791} C_DIS
LIN {X 96.3294,Y -98.529,Z 179,A -41.7354,B 5.6394,C 0.3394,E1 5.7633,E2 494.0433} C_DIS
LIN {X 99.3091,Y -95.5258,Z 179,A -40.0328,B 5.6396,C 0.3366,E1 5.7666,E2 492.3465} C_DIS
LIN {X 101.9011,Y -92.7549,Z 179,A -38.4617,B 5.6398,C 0.3333,E1 5.7696,E2 490.7748} C_DIS
LIN {X 104.6983,Y -89.5864,Z 179,A -36.7626,B 5.6399,C 0.3303,E1 5.7727,E2 489.0819} C_DIS
LIN {X 107.4763,Y -86.2336,Z 179,A -35.0334,B 5.6401,C 0.3274,E1 5.7757,E2 487.3617} C_DIS
LIN {X 109.722,Y -83.358,Z 179,A -33.5034,B 5.6403,C 0.3237,E1 5.7783,E2 485.8286} C_DIS
LIN {X 111.9633,Y -80.3215,Z 179,A -31.9439,B 5.6405,C 0.3201,E1 5.7809,E2 484.269} C_DIS
LIN {X 114.4304,Y -76.7663,Z 179,A -30.1569,B 5.6408,C 0.316,E1 5.7837,E2 482.482} C_DIS
LIN {X 116.8847,Y -72.9746,Z 179,A -28.3499,B 5.641,C 0.3125,E1 5.7864,E2 480.6825} C_DIS
LIN {X 119.0333,Y -69.4157,Z 179,A -26.6386,B 5.6412,C 0.3084,E1 5.7888,E2 478.972} C_DIS
LIN {X 121.1775,Y -65.6009,Z 179,A -24.955,B 5.6413,C 0.3059,E1 5.7911,E2 477.3044} C_DIS
LIN {X 122.6031,Y -62.8917,Z 179,A -23.8739,B 5.6413,C 0.3056,E1 5.7924,E2 476.247} C_DIS
LIN {X 123.9586,Y -60.1808,Z 179,A -22.4837,B 5.6416,C 0.3003,E1 5.7942,E2 474.8388} C_DIS
LIN {X 125.6114,Y -56.6453,Z 179,A -21.058,B 5.6416,C 0.2992,E1 5.7958,E2 473.4372} C_DIS
LIN {X 126.8184,Y -53.894,Z 179,A -19.6808,B 5.6419,C 0.2939,E1 5.7974,E2 472.0423} C_DIS
Enddeposition()
END
